KUKA KRL program: MyProgram_194().src

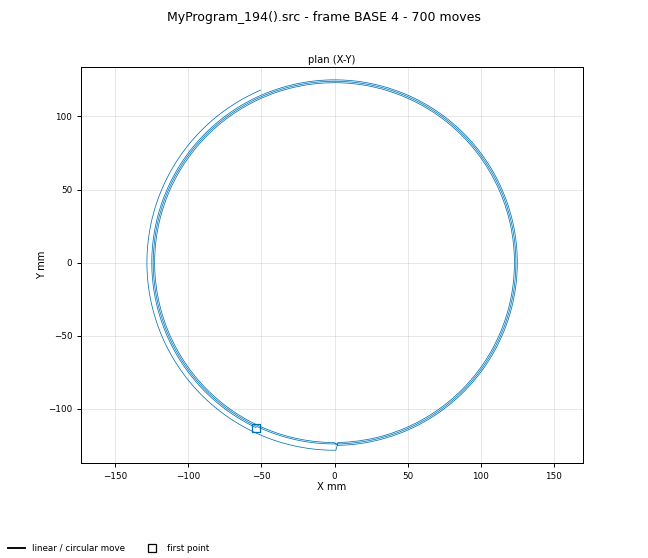
[picture p0: tool path of MyProgram_194().src in frame BASE 4, 700 of 700 moves have a stored position in this frame; points joined in program order, loops and branches not executed]
&ACCESS RVP
&REL 1
&PARAM TEMPLATE = C:\KRC\Roboter\Template\vorgabe
&PARAM EDITMASK = *
DEF MyProgram_194()
; ---- Setting reference (Base) ----
$BASE = BASE_DATA[4]

; --------------------------
; ---- Setting tool (TCP) ----
$TOOL = TOOL_DATA[3]
; --------------------------

$VEL.CP = VEL_APROX_PRINT
Startdeposition()
$VEL.CP = VEL_PRINT
LIN {X -53.6919,Y -112.9399,Z 140,A -118.7659,B 24.3079,C -1.2792,E1 24.2705,E2 205.3215} C_DIS
LIN {X -56.5912,Y -111.5152,Z 140,A -120.1079,B 24.3075,C -1.2873,E1 24.2671,E2 206.6473} C_DIS
LIN {X -59.8719,Y -109.7908,Z 140,A -122.1119,B 24.3081,C -1.2756,E1 24.2621,E2 208.6856} C_DIS
LIN {X -63.0275,Y -108.0107,Z 140,A -124.4326,B 24.3094,C -1.2483,E1 24.2563,E2 211.08} C_DIS
LIN {X -67.2513,Y -105.4322,Z 140,A -126.1298,B 24.308,C -1.2774,E1 24.2525,E2 212.7119} C_DIS
LIN {X -70.1428,Y -103.5309,Z 140,A -127.4855,B 24.3074,C -1.2903,E1 24.2494,E2 214.0408} C_DIS
LIN {X -72.9333,Y -101.5847,Z 140,A -129.2817,B 24.3078,C -1.2823,E1 24.2452,E2 215.8629} C_DIS
LIN {X -76.3639,Y -99.0319,Z 140,A -131.2624,B 24.3076,C -1.2848,E1 24.2408,E2 217.8448} C_DIS
LIN {X -79.5467,Y -96.4938,Z 140,A -133.1846,B 24.3076,C -1.2858,E1 24.2366,E2 219.7721} C_DIS
LIN {X -83.0381,Y -93.5062,Z 140,A -135.2359,B 24.3072,C -1.2924,E1 24.2323,E2 221.8156} C_DIS
LIN {X -86.157,Y -90.6407,Z 140,A -137.2143,B 24.3072,C -1.2947,E1 24.2283,E2 223.7967} C_DIS
LIN {X -89.322,Y -87.5228,Z 140,A -139.2228,B 24.3069,C -1.3003,E1 24.2243,E2 225.8004} C_DIS
LIN {X -91.6108,Y -85.1243,Z 140,A -140.6773,B 24.3065,C -1.3065,E1 24.2216,E2 227.2461} C_DIS
LIN {X -95.1006,Y -81.2071,Z 140,A -143.1881,B 24.3065,C -1.3073,E1 24.2169,E2 229.7666} C_DIS
LIN {X -97.6117,Y -78.1712,Z 140,A -145.009,B 24.3063,C -1.311,E1 24.2137,E2 231.5874} C_DIS
LIN {X -100.1442,Y -74.8991,Z 140,A -146.9149,B 24.3061,C -1.3152,E1 24.2105,E2 233.4924} C_DIS
LIN {X -102.2447,Y -72.0048,Z 140,A -148.8726,B 24.3066,C -1.3054,E1 24.2073,E2 235.4839} C_DIS
LIN {X -104.3595,Y -68.9041,Z 140,A -150.5706,B 24.3063,C -1.3108,E1 24.2047,E2 237.1775} C_DIS
LIN {X -106.3024,Y -65.8673,Z 140,A -151.9331,B 24.3055,C -1.3278,E1 24.2027,E2 238.5057} C_DIS
LIN {X -108.4877,Y -62.2025,Z 140,A -153.9183,B 24.3053,C -1.3317,E1 24.1999,E2 240.4918} C_DIS
LIN {X -110.5462,Y -58.4624,Z 140,A -155.833,B 24.3049,C -1.339,E1 24.1974,E2 242.3992} C_DIS
LIN {X -112.655,Y -54.2883,Z 140,A -158.0264,B 24.3047,C -1.3428,E1 24.1947,E2 244.5954} C_DIS
LIN {X -113.9621,Y -51.4883,Z 140,A -159.552,B 24.3047,C -1.3421,E1 24.1929,E2 246.1313} C_DIS
LIN {X -115.8635,Y -47.0528,Z 140,A -161.597,B 24.304,C -1.3558,E1 24.1907,E2 248.1546} C_DIS
LIN {X -117.0482,Y -44.0221,Z 140,A -163.0377,B 24.3037,C -1.3624,E1 24.1893,E2 249.5876} C_DIS
LIN {X -118.0271,Y -41.3277,Z 140,A -164.4301,B 24.3037,C -1.3629,E1 24.188,E2 250.9868} C_DIS
LIN {X -119.0708,Y -38.2151,Z 140,A -165.9048,B 24.3033,C -1.3688,E1 24.1867,E2 252.456} C_DIS
LIN {X -120.7278,Y -32.6066,Z 140,A -168.6751,B 24.3031,C -1.3731,E1 24.1845,E2 255.2322} C_DIS
LIN {X -121.683,Y -28.8394,Z 140,A -171.0654,B 24.3042,C -1.3525,E1 24.183,E2 257.6873} C_DIS
LIN {X -122.7191,Y -24.0546,Z 140,A -172.5557,B 24.3021,C -1.3918,E1 24.1822,E2 259.0906} C_DIS
LIN {X -123.7321,Y -18.1343,Z 140,A -175.4845,B 24.3021,C -1.3929,E1 24.1808,E2 262.0347} C_DIS
LIN {X -124.1912,Y -14.6583,Z 140,A -177.2858,B 24.3022,C -1.3897,E1 24.1802,E2 263.8548} C_DIS
LIN {X -124.6891,Y -9.5463,Z 140,A -179.4863,B 24.3014,C -1.4038,E1 24.1797,E2 266.0345} C_DIS
LIN {X -124.93,Y -5.5935,Z 140,A 178.647,B 24.3012,C -1.4075,E1 24.1794,E2 267.9039} C_DIS
LIN {X -125.0405,Y -1.8059,Z 140,A 177.1827,B 24.3003,C -1.4248,E1 24.1793,E2 269.3348} C_DIS
LIN {X -125.0536,Y 0.6006,Z 140,A 175.2536,B 24.302,C -1.3931,E1 24.1793,E2 271.3536} C_DIS
LIN {X -124.9418,Y 5.2951,Z 140,A 173.618,B 24.3004,C -1.4221,E1 24.1795,E2 272.9285} C_DIS
LIN {X -124.7099,Y 9.2612,Z 140,A 171.2259,B 24.3014,C -1.4037,E1 24.18,E2 275.3803} C_DIS
LIN {X -124.2464,Y 14.1956,Z 140,A 169.6952,B 24.2993,C -1.4426,E1 24.1804,E2 276.8253} C_DIS
LIN {X -123.3534,Y 20.5476,Z 140,A 166.6428,B 24.299,C -1.4473,E1 24.1817,E2 279.8851} C_DIS
LIN {X -122.8031,Y 23.6152,Z 140,A 165.0229,B 24.2992,C -1.4437,E1 24.1825,E2 281.5236} C_DIS
LIN {X -121.7214,Y 28.6802,Z 140,A 162.7251,B 24.2986,C -1.4545,E1 24.1839,E2 283.8089} C_DIS
LIN {X -120.7968,Y 32.3479,Z 140,A 161.1059,B 24.2981,C -1.465,E1 24.185,E2 285.4122} C_DIS
LIN {X -119.8901,Y 35.5638,Z 140,A 159.5609,B 24.2978,C -1.4692,E1 24.1862,E2 286.956} C_DIS
LIN {X -118.4982,Y 39.9577,Z 140,A 157.3573,B 24.2977,C -1.472,E1 24.1881,E2 289.166} C_DIS
LIN {X -117.1953,Y 43.6296,Z 140,A 155.618,B 24.2972,C -1.4795,E1 24.1897,E2 290.8969} C_DIS
LIN {X -115.9948,Y 46.7269,Z 140,A 153.9199,B 24.2974,C -1.4767,E1 24.1915,E2 292.6117} C_DIS
LIN {X -114.7571,Y 49.6891,Z 140,A 152.2718,B 24.2976,C -1.4736,E1 24.1934,E2 294.2767} C_DIS
LIN {X -113.4363,Y 52.6348,Z 140,A 150.9968,B 24.2968,C -1.4869,E1 24.1948,E2 295.5265} C_DIS
LIN {X -111.6462,Y 56.3339,Z 140,A 149.1355,B 24.2964,C -1.4934,E1 24.1971,E2 297.3821} C_DIS
LIN {X -110.3342,Y 58.8656,Z 140,A 147.8595,B 24.2961,C -1.4986,E1 24.1988,E2 298.6525} C_DIS
LIN {X -108.0224,Y 63.0061,Z 140,A 145.4957,B 24.2962,C -1.4968,E1 24.2021,E2 301.0336} C_DIS
LIN {X -105.5652,Y 67.043,Z 140,A 143.405,B 24.2957,C -1.5062,E1 24.2051,E2 303.1123} C_DIS
LIN {X -103.2652,Y 70.5339,Z 140,A 141.529,B 24.2953,C -1.5133,E1 24.208,E2 304.9806} C_DIS
LIN {X -101.1094,Y 73.5907,Z 140,A 139.7773,B 24.2951,C -1.5164,E1 24.2109,E2 306.7335} C_DIS
LIN {X -98.532,Y 77.0078,Z 140,A 137.7937,B 24.2948,C -1.5207,E1 24.2143,E2 308.7163} C_DIS
LIN {X -95.8068,Y 80.3723,Z 140,A 135.8162,B 24.2945,C -1.5262,E1 24.2178,E2 310.6897} C_DIS
LIN {X -92.9689,Y 83.6392,Z 140,A 133.8174,B 24.2942,C -1.5306,E1 24.2214,E2 312.6871} C_DIS
LIN {X -90.0744,Y 86.7489,Z 140,A 131.8247,B 24.2941,C -1.5334,E1 24.2253,E2 314.6818} C_DIS
LIN {X -86.8221,Y 90.0035,Z 140,A 129.7974,B 24.2936,C -1.5421,E1 24.2293,E2 316.6968} C_DIS
LIN {X -83.7569,Y 92.8632,Z 140,A 127.7843,B 24.2936,C -1.5425,E1 24.2334,E2 318.7171} C_DIS
LIN {X -80.5197,Y 95.6832,Z 140,A 125.8611,B 24.2932,C -1.5489,E1 24.2375,E2 320.6324} C_DIS
LIN {X -77.3248,Y 98.2829,Z 140,A 123.9446,B 24.293,C -1.5518,E1 24.2417,E2 322.5494} C_DIS
LIN {X -73.8783,Y 100.8994,Z 140,A 121.9198,B 24.2928,C -1.5541,E1 24.2462,E2 324.576} C_DIS
LIN {X -70.4181,Y 103.3445,Z 140,A 119.9558,B 24.2927,C -1.557,E1 24.2507,E2 326.5399} C_DIS
LIN {X -66.6736,Y 105.7984,Z 140,A 117.95,B 24.2923,C -1.5629,E1 24.2554,E2 328.5378} C_DIS
LIN {X -63.9124,Y 107.489,Z 140,A 116.1645,B 24.293,C -1.5524,E1 24.2598,E2 330.3547} C_DIS
LIN {X -60.9161,Y 109.2142,Z 140,A 114.5683,B 24.2928,C -1.5546,E1 24.2637,E2 331.9502} C_DIS
LIN {X -57.8736,Y 110.8554,Z 140,A 113.5124,B 24.2912,C -1.5807,E1 24.2661,E2 332.9456} C_DIS
LIN {X -54.8742,Y 112.3711,Z 140,A 111.3515,B 24.2928,C -1.5556,E1 24.2717,E2 335.1734} C_DIS
LIN {X -51.3522,Y 114.023,Z 140,A 109.9613,B 24.2915,C -1.5757,E1 24.2751,E2 336.5181} C_DIS
LIN {X -47.4788,Y 115.6917,Z 140,A 107.9839,B 24.2915,C -1.5764,E1 24.2802,E2 338.4984} C_DIS
LIN {X -44.6099,Y 116.8278,Z 140,A 106.6024,B 24.2913,C -1.5798,E1 24.2838,E2 339.8748} C_DIS
LIN {X -41.6192,Y 117.9259,Z 140,A 104.3148,B 24.2934,C -1.5449,E1 24.2901,E2 342.252} C_DIS
LIN {X -35.9049,Y 119.7898,Z 140,A 102.3187,B 24.2912,C -1.5817,E1 24.2952,E2 344.1621} C_DIS
LIN {X -32.8305,Y 120.6681,Z 140,A 100.5146,B 24.292,C -1.568,E1 24.3001,E2 346.0023} C_DIS
LIN {X -29.118,Y 121.6159,Z 140,A 98.6999,B 24.292,C -1.567,E1 24.3051,E2 347.822} C_DIS
LIN {X -25.0294,Y 122.5226,Z 140,A 97.2935,B 24.2906,C -1.5917,E1 24.3088,E2 349.1699} C_DIS
LIN {X -21.6294,Y 123.169,Z 140,A 95.5831,B 24.2908,C -1.5873,E1 24.3135,E2 350.893} C_DIS
LIN {X -17.7649,Y 123.7849,Z 140,A 93.8925,B 24.2905,C -1.5931,E1 24.3181,E2 352.5708} C_DIS
LIN {X -13.8843,Y 124.281,Z 140,A 92.0908,B 24.2905,C -1.5937,E1 24.3231,E2 354.3723} C_DIS
LIN {X -10.2183,Y 124.6354,Z 140,A 90.3228,B 24.2906,C -1.5909,E1 24.328,E2 356.1481} C_DIS
LIN {X -6.2274,Y 124.8981,Z 140,A 88.5896,B 24.2903,C -1.5961,E1 24.3328,E2 357.8691} C_DIS
LIN {X -2.719,Y 125.0254,Z 140,A 86.9015,B 24.2905,C -1.5929,E1 24.3376,E2 359.5653} C_DIS
LIN {X 1.0171,Y 125.0496,Z 140,A 85.1762,B 24.2905,C -1.5926,E1 24.3424,E2 361.2912} C_DIS
LIN {X 4.9283,Y 124.9561,Z 140,A 83.4543,B 24.2903,C -1.596,E1 24.3472,E2 363.0044} C_DIS
LIN {X 8.9204,Y 124.7348,Z 140,A 81.6298,B 24.2903,C -1.5964,E1 24.3523,E2 364.8273} C_DIS
LIN {X 12.4955,Y 124.4285,Z 140,A 79.8894,B 24.2906,C -1.5917,E1 24.3571,E2 366.5781} C_DIS
LIN {X 16.3314,Y 123.9821,Z 140,A 78.2129,B 24.2903,C -1.5956,E1 24.3617,E2 368.2436} C_DIS
LIN {X 20.3658,Y 123.3838,Z 140,A 76.3517,B 24.2903,C -1.5954,E1 24.3669,E2 370.1036} C_DIS
LIN {X 24.186,Y 122.694,Z 140,A 74.372,B 24.291,C -1.5853,E1 24.3724,E2 372.1055} C_DIS
LIN {X 29.3374,Y 121.563,Z 140,A 72.182,B 24.2904,C -1.5946,E1 24.3783,E2 374.2698} C_DIS
LIN {X 32.964,Y 120.6323,Z 140,A 70.3195,B 24.2909,C -1.5865,E1 24.3833,E2 376.1488} C_DIS
LIN {X 36.874,Y 119.4932,Z 140,A 68.5454,B 24.2907,C -1.5894,E1 24.388,E2 377.9126} C_DIS
LIN {X 40.4587,Y 118.3283,Z 140,A 66.9207,B 24.2905,C -1.5928,E1 24.3923,E2 379.526} C_DIS
LIN {X 43.1079,Y 117.3901,Z 140,A 65.0136,B 24.2923,C -1.5624,E1 24.3975,E2 381.5026} C_DIS
LIN {X 47.2438,Y 115.7865,Z 140,A 63.4562,B 24.2911,C -1.5827,E1 24.4014,E2 383.0074} C_DIS
LIN {X 50.698,Y 114.3156,Z 140,A 61.8125,B 24.2911,C -1.5844,E1 24.4056,E2 384.6428} C_DIS
LIN {X 54.3579,Y 112.6217,Z 140,A 59.6104,B 24.2922,C -1.5653,E1 24.4112,E2 386.8852} C_DIS
LIN {X 57.603,Y 110.9975,Z 140,A 58.2793,B 24.2913,C -1.5788,E1 24.4145,E2 388.1797} C_DIS
LIN {X 63.6338,Y 107.6546,Z 140,A 55.1206,B 24.2916,C -1.5743,E1 24.4222,E2 391.3398} C_DIS
LIN {X 67.1422,Y 105.5021,Z 140,A 53.3746,B 24.2914,C -1.578,E1 24.4262,E2 393.0709} C_DIS
LIN {X 70.2121,Y 103.484,Z 140,A 51.6783,B 24.2916,C -1.5746,E1 24.4302,E2 394.7697} C_DIS
LIN {X 73.1481,Y 101.4302,Z 140,A 50.0018,B 24.2919,C -1.5701,E1 24.434,E2 396.4511} C_DIS
LIN {X 76.1718,Y 99.1795,Z 140,A 48.3051,B 24.2919,C -1.5685,E1 24.4378,E2 398.1456} C_DIS
LIN {X 80.5194,Y 95.6834,Z 140,A 45.661,B 24.2925,C -1.5593,E1 24.4436,E2 400.8015} C_DIS
LIN {X 83.7682,Y 92.8529,Z 140,A 43.6395,B 24.2929,C -1.553,E1 24.4478,E2 402.8298} C_DIS
LIN {X 87.085,Y 89.7489,Z 140,A 41.6152,B 24.293,C -1.5514,E1 24.4519,E2 404.8495} C_DIS
LIN {X 90.0335,Y 86.7911,Z 140,A 39.6982,B 24.2933,C -1.547,E1 24.4556,E2 406.7686} C_DIS
LIN {X 92.8649,Y 83.755,Z 140,A 37.7842,B 24.2936,C -1.5421,E1 24.4592,E2 408.6858} C_DIS
LIN {X 95.6504,Y 80.5588,Z 140,A 35.8982,B 24.2936,C -1.5403,E1 24.4627,E2 410.5672} C_DIS
LIN {X 98.1158,Y 77.5376,Z 140,A 34.0944,B 24.294,C -1.5352,E1 24.4658,E2 412.3749} C_DIS
LIN {X 100.6643,Y 74.1983,Z 140,A 32.3122,B 24.2938,C -1.5374,E1 24.4688,E2 414.1431} C_DIS
LIN {X 103.2862,Y 70.5033,Z 140,A 30.1538,B 24.2944,C -1.528,E1 24.4723,E2 416.3133} C_DIS
LIN {X 105.5787,Y 67.0216,Z 140,A 28.1882,B 24.2949,C -1.5202,E1 24.4753,E2 418.2874} C_DIS
LIN {X 107.2835,Y 64.2572,Z 140,A 26.4298,B 24.2959,C -1.5029,E1 24.4778,E2 420.0784} C_DIS
LIN {X 109.1198,Y 61.0865,Z 140,A 25.055,B 24.2953,C -1.5132,E1 24.4797,E2 421.4208} C_DIS
LIN {X 110.6437,Y 58.2767,Z 140,A 23.1393,B 24.2968,C -1.487,E1 24.4822,E2 423.3896} C_DIS
LIN {X 112.6736,Y 54.2493,Z 140,A 21.7292,B 24.2953,C -1.5134,E1 24.4839,E2 424.728} C_DIS
LIN {X 114.1511,Y 51.0659,Z 140,A 20.0748,B 24.2957,C -1.5065,E1 24.4858,E2 426.3899} C_DIS
LIN {X 115.3595,Y 48.2741,Z 140,A 18.7408,B 24.2957,C -1.5054,E1 24.4873,E2 427.7191} C_DIS
LIN {X 116.3256,Y 45.9017,Z 140,A 17.4038,B 24.2964,C -1.4938,E1 24.4887,E2 429.0764} C_DIS
LIN {X 117.9032,Y 41.6849,Z 140,A 14.9511,B 24.2979,C -1.4683,E1 24.491,E2 431.5767} C_DIS
LIN {X 119.1859,Y 37.8547,Z 140,A 13.4947,B 24.2971,C -1.4822,E1 24.4922,E2 432.991} C_DIS
LIN {X 120.8839,Y 32.0214,Z 140,A 10.8374,B 24.2972,C -1.4799,E1 24.4943,E2 435.6381} C_DIS
LIN {X 121.8046,Y 28.3208,Z 140,A 9.1135,B 24.2974,C -1.4756,E1 24.4954,E2 437.3621} C_DIS
LIN {X 122.5443,Y 24.923,Z 140,A 7.5415,B 24.2977,C -1.4716,E1 24.4963,E2 438.9342} C_DIS
LIN {X 123.2508,Y 21.1628,Z 140,A 5.724,B 24.2982,C -1.4628,E1 24.4972,E2 440.7621} C_DIS
LIN {X 123.8051,Y 17.6236,Z 140,A 4.1393,B 24.2983,C -1.4604,E1 24.4978,E2 442.343} C_DIS
LIN {X 124.3134,Y 13.5837,Z 140,A 2.3029,B 24.2986,C -1.4558,E1 24.4985,E2 444.1792} C_DIS
LIN {X 124.6751,Y 9.7384,Z 140,A 0.4725,B 24.2991,C -1.447,E1 24.4989,E2 446.0197} C_DIS
LIN {X 124.9132,Y 5.9267,Z 140,A -1.2863,B 24.2994,C -1.4409,E1 24.4992,E2 447.7825} C_DIS
LIN {X 125.0374,Y 1.9942,Z 140,A -2.9417,B 24.2994,C -1.4424,E1 24.4992,E2 449.4241} C_DIS
LIN {X 125.0322,Y -2.3088,Z 140,A -5.0331,B 24.3,C -1.43,E1 24.4992,E2 451.5328} C_DIS
LIN {X 124.8915,Y -6.358,Z 140,A -6.7859,B 24.3,C -1.4291,E1 24.499,E2 453.2769} C_DIS
LIN {X 124.6624,Y -9.8989,Z 140,A -8.4794,B 24.3005,C -1.4203,E1 24.4987,E2 454.9812} C_DIS
LIN {X 124.3069,Y -13.644,Z 140,A -10.2178,B 24.3009,C -1.414,E1 24.4982,E2 456.7244} C_DIS
LIN {X 123.7958,Y -17.688,Z 140,A -11.9726,B 24.3009,C -1.4135,E1 24.4975,E2 458.4695} C_DIS
LIN {X 123.1515,Y -21.7273,Z 140,A -13.8398,B 24.3012,C -1.4078,E1 24.4967,E2 460.3394} C_DIS
LIN {X 121.8901,Y -27.9473,Z 140,A -17.1147,B 24.3027,C -1.38,E1 24.4947,E2 463.6617} C_DIS
LIN {X 120.9852,Y -31.6414,Z 140,A -18.357,B 24.3017,C -1.3994,E1 24.4939,E2 464.8498} C_DIS
LIN {X 120.1853,Y -34.5514,Z 140,A -20.0597,B 24.3028,C -1.379,E1 24.4926,E2 466.5918} C_DIS
LIN {X 118.7173,Y -39.2996,Z 140,A -22.4113,B 24.3034,C -1.368,E1 24.4906,E2 468.9561} C_DIS
LIN {X 117.6172,Y -42.4784,Z 140,A -23.603,B 24.3027,C -1.3806,E1 24.4895,E2 470.1105} C_DIS
LIN {X 116.369,Y -45.79,Z 140,A -25.192,B 24.3029,C -1.3772,E1 24.4879,E2 471.6988} C_DIS
LIN {X 115.0127,Y -49.098,Z 140,A -26.9146,B 24.3034,C -1.3678,E1 24.486,E2 473.4341} C_DIS
LIN {X 112.0407,Y -55.544,Z 140,A -30.0975,B 24.3037,C -1.3614,E1 24.4822,E2 476.6149} C_DIS
LIN {X 109.9969,Y -59.4933,Z 140,A -32.1786,B 24.3041,C -1.3531,E1 24.4795,E2 478.7047} C_DIS
LIN {X 108.034,Y -62.9877,Z 140,A -34.0489,B 24.3045,C -1.346,E1 24.4769,E2 480.5823} C_DIS
LIN {X 105.6721,Y -66.8737,Z 140,A -36.0672,B 24.3047,C -1.3432,E1 24.4739,E2 482.5967} C_DIS
LIN {X 102.7414,Y -71.2944,Z 140,A -38.3754,B 24.3047,C -1.3424,E1 24.4704,E2 484.8951} C_DIS
LIN {X 100.5448,Y -74.361,Z 140,A -40.2595,B 24.3054,C -1.3298,E1 24.4672,E2 486.8001} C_DIS
LIN {X 97.8823,Y -77.8313,Z 140,A -42.2174,B 24.3055,C -1.3267,E1 24.4639,E2 488.7562} C_DIS
LIN {X 94.2467,Y -82.1962,Z 140,A -44.7886,B 24.3058,C -1.3214,E1 24.4592,E2 491.328} C_DIS
LIN {X 89.1498,Y -87.6983,Z 140,A -48.0245,B 24.3058,C -1.3226,E1 24.4531,E2 494.5465} C_DIS
LIN {X 85.4413,Y -91.3155,Z 140,A -50.5983,B 24.3065,C -1.3069,E1 24.4478,E2 497.1472} C_DIS
LIN {X 80.2995,Y -95.8679,Z 140,A -53.7377,B 24.3069,C -1.3,E1 24.4412,E2 500.2906} C_DIS
LIN {X 76.9147,Y -98.6049,Z 140,A -55.7259,B 24.3071,C -1.2959,E1 24.4369,E2 502.2812} C_DIS
LIN {X 73.3148,Y -101.3095,Z 140,A -57.4223,B 24.3064,C -1.3095,E1 24.4332,E2 503.9382} C_DIS
LIN {X 68.4944,Y -104.6293,Z 140,A -60.4164,B 24.3074,C -1.2887,E1 24.4262,E2 506.9722} C_DIS
LIN {X 64.8243,Y -106.9415,Z 140,A -62.3627,B 24.3075,C -1.2869,E1 24.4215,E2 508.9166} C_DIS
LIN {X 61.0777,Y -109.1248,Z 140,A -64.375,B 24.3078,C -1.2821,E1 24.4166,E2 510.9344} C_DIS
LIN {X 57.1048,Y -111.2538,Z 140,A -66.3773,B 24.3078,C -1.2816,E1 24.4117,E2 512.9321} C_DIS
LIN {X 54.2085,Y -112.6931,Z 140,A -67.7822,B 24.3078,C -1.2829,E1 24.4082,E2 514.3299} C_DIS
LIN {X 51.3542,Y -114.0221,Z 140,A -69.338,B 24.3081,C -1.2752,E1 24.4042,E2 515.9004} C_DIS
LIN {X 47.6413,Y -115.6238,Z 140,A -71.2144,B 24.3083,C -1.2713,E1 24.3994,E2 517.7817} C_DIS
LIN {X 44.1737,Y -116.9914,Z 140,A -73.5929,B 24.31,C -1.2368,E1 24.393,E2 520.2386} C_DIS
LIN {X 38.856,Y -118.865,Z 140,A -75.3361,B 24.3082,C -1.2737,E1 24.3886,E2 521.8887} C_DIS
LIN {X 32.1785,Y -120.842,Z 140,A -78.5471,B 24.3084,C -1.2691,E1 24.38,E2 525.1052} C_DIS
LIN {X 28.7784,Y -121.6977,Z 140,A -80.1455,B 24.3084,C -1.2679,E1 24.3756,E2 526.7042} C_DIS
LIN {X 24.9652,Y -122.5357,Z 140,A -81.941,B 24.3086,C -1.266,E1 24.3707,E2 528.502} C_DIS
LIN {X 21.4154,Y -123.2073,Z 140,A -83.6474,B 24.3087,C -1.2622,E1 24.366,E2 530.2157} C_DIS
LIN {X 17.7573,Y -123.7859,Z 140,A -85.2968,B 24.3087,C -1.2633,E1 24.3615,E2 531.8608} C_DIS
LIN {X 14.0315,Y -124.2652,Z 140,A -87.0869,B 24.3089,C -1.2589,E1 24.3565,E2 533.6602} C_DIS
LIN {X 10.4122,Y -124.619,Z 140,A -88.6895,B 24.3088,C -1.2611,E1 24.352,E2 535.2565} C_DIS
LIN {X 6.4833,Y -124.8852,Z 140,A -90.5192,B 24.3088,C -1.2591,E1 24.3469,E2 537.0903} C_DIS
LIN {X 2.4731,Y -125.0294,Z 140,A -92.3766,B 24.309,C -1.2576,E1 24.3417,E2 538.9509} C_DIS
LIN {X 2.4731,Y -125.0294,Z 140,A -92.3766,B 24.309,C -1.2576,E1 24.3417,E2 538.9509} C_DIS
Enddeposition()
LIN {X 0.8758,Y -124.0739,Z 140,A -92.8769,B 23.7005,C -1.164,E1 23.7279,E2 539.5997} C_DIS
Startdeposition()
$VEL.CP = VEL_PRINT
LIN {X 5.1874,Y -123.9703,Z 140,A -90.2212,B 23.6991,C -1.195,E1 23.7355,E2 536.8673} C_DIS
LIN {X 8.9976,Y -123.7516,Z 140,A -88.3652,B 23.6989,C -1.2001,E1 23.7407,E2 534.9995} C_DIS
LIN {X 13.0801,Y -123.387,Z 140,A -86.5046,B 23.6989,C -1.1996,E1 23.7459,E2 533.1412} C_DIS
LIN {X 16.4159,Y -122.9878,Z 140,A -84.9017,B 23.6987,C -1.203,E1 23.7503,E2 531.5313} C_DIS
LIN {X 20.3643,Y -122.3956,Z 140,A -83.1274,B 23.6988,C -1.2011,E1 23.7552,E2 529.7636} C_DIS
LIN {X 23.38,Y -121.8554,Z 140,A -81.6488,B 23.6986,C -1.2053,E1 23.7593,E2 528.2764} C_DIS
LIN {X 27.1976,Y -121.0613,Z 140,A -79.4825,B 23.6977,C -1.2241,E1 23.7653,E2 526.0664} C_DIS
LIN {X 30.9893,Y -120.1468,Z 140,A -78.0716,B 23.6985,C -1.2075,E1 23.769,E2 524.699} C_DIS
LIN {X 38.5918,Y -117.9254,Z 140,A -74.5759,B 23.6987,C -1.204,E1 23.7783,E2 521.2185} C_DIS
LIN {X 43.8221,Y -116.0821,Z 140,A -71.9287,B 23.6983,C -1.2115,E1 23.7853,E2 518.5586} C_DIS
LIN {X 46.5763,Y -115.0043,Z 140,A -70.4957,B 23.6981,C -1.2166,E1 23.789,E2 517.1163} C_DIS
LIN {X 49.8037,Y -113.6454,Z 140,A -69.0055,B 23.6982,C -1.2129,E1 23.7928,E2 515.639} C_DIS
LIN {X 52.648,Y -112.356,Z 140,A -67.5899,B 23.6982,C -1.2139,E1 23.7964,E2 514.2247} C_DIS
LIN {X 55.0194,Y -111.2123,Z 140,A -66.3236,B 23.698,C -1.2183,E1 23.7996,E2 512.951} C_DIS
LIN {X 58.3255,Y -109.5169,Z 140,A -64.508,B 23.6976,C -1.226,E1 23.8041,E2 511.1218} C_DIS
LIN {X 61.5286,Y -107.7497,Z 140,A -62.8692,B 23.6976,C -1.2266,E1 23.8081,E2 509.4866} C_DIS
LIN {X 64.6525,Y -105.9051,Z 140,A -61.2958,B 23.6976,C -1.2248,E1 23.8119,E2 507.9229} C_DIS
LIN {X 67.6259,Y -104.0312,Z 140,A -59.657,B 23.6975,C -1.2287,E1 23.8157,E2 506.2801} C_DIS
LIN {X 71.3355,Y -101.5236,Z 140,A -57.7263,B 23.6975,C -1.2263,E1 23.8202,E2 504.3623} C_DIS
LIN {X 73.7735,Y -99.7666,Z 140,A -56.07,B 23.6968,C -1.2421,E1 23.824,E2 502.673} C_DIS
LIN {X 77.3218,Y -97.0418,Z 140,A -54.0651,B 23.6968,C -1.2437,E1 23.8284,E2 500.6721} C_DIS
LIN {X 80.6334,Y -94.3082,Z 140,A -52.0635,B 23.6965,C -1.2491,E1 23.8326,E2 498.6653} C_DIS
LIN {X 82.9928,Y -92.239,Z 140,A -50.6939,B 23.6965,C -1.2486,E1 23.8355,E2 497.3027} C_DIS
LIN {X 86.0033,Y -89.4389,Z 140,A -48.7547,B 23.6962,C -1.2551,E1 23.8394,E2 495.356} C_DIS
LIN {X 89.6603,Y -85.7716,Z 140,A -46.2997,B 23.6957,C -1.2641,E1 23.8442,E2 492.8898} C_DIS
LIN {X 91.9569,Y -83.3048,Z 140,A -44.8695,B 23.6958,C -1.2619,E1 23.8469,E2 491.4717} C_DIS
LIN {X 94.4731,Y -80.44,Z 140,A -43.0875,B 23.6955,C -1.2675,E1 23.8502,E2 489.6843} C_DIS
LIN {X 97.9235,Y -76.2024,Z 140,A -40.7829,B 23.6957,C -1.2636,E1 23.8542,E2 487.4009} C_DIS
LIN {X 99.712,Y -73.847,Z 140,A -39.363,B 23.6954,C -1.2699,E1 23.8566,E2 485.9725} C_DIS
LIN {X 101.7025,Y -71.0805,Z 140,A -37.6313,B 23.6948,C -1.282,E1 23.8594,E2 484.2198} C_DIS
LIN {X 103.8864,Y -67.849,Z 140,A -35.8252,B 23.6945,C -1.2873,E1 23.8622,E2 482.4101} C_DIS
LIN {X 106.1614,Y -64.2301,Z 140,A -33.964,B 23.6945,C -1.2875,E1 23.8649,E2 480.5584} C_DIS
LIN {X 108.1442,Y -60.8325,Z 140,A -32.0915,B 23.6941,C -1.2956,E1 23.8675,E2 478.6763} C_DIS
LIN {X 110.0019,Y -57.4018,Z 140,A -30.3709,B 23.6941,C -1.297,E1 23.8698,E2 476.9618} C_DIS
LIN {X 112.2352,Y -52.9053,Z 140,A -28.1101,B 23.6938,C -1.3011,E1 23.8725,E2 474.7037} C_DIS
LIN {X 113.4448,Y -50.2572,Z 140,A -26.8255,B 23.6938,C -1.3023,E1 23.874,E2 473.4236} C_DIS
LIN {X 114.84,Y -46.9841,Z 140,A -25.2021,B 23.6936,C -1.3064,E1 23.8757,E2 471.7995} C_DIS
LIN {X 115.7727,Y -44.633,Z 140,A -23.8604,B 23.6929,C -1.3185,E1 23.8771,E2 470.4356} C_DIS
LIN {X 117.0146,Y -41.2717,Z 140,A -22.2604,B 23.6928,C -1.321,E1 23.8786,E2 468.839} C_DIS
LIN {X 118.1823,Y -37.7925,Z 140,A -20.5905,B 23.6926,C -1.3251,E1 23.8801,E2 467.1689} C_DIS
LIN {X 119.6482,Y -32.863,Z 140,A -18.3162,B 23.6924,C -1.3277,E1 23.8818,E2 464.902} C_DIS
LIN {X 120.5452,Y -29.3992,Z 140,A -15.7166,B 23.6896,C -1.3799,E1 23.8836,E2 462.1891} C_DIS
LIN {X 121.8513,Y -23.4014,Z 140,A -14.1238,B 23.6924,C -1.3276,E1 23.8845,E2 460.7356} C_DIS
LIN {X 122.5522,Y -19.4042,Z 140,A -11.9092,B 23.6912,C -1.3504,E1 23.8855,E2 458.4786} C_DIS
LIN {X 123.0592,Y -15.871,Z 140,A -10.2349,B 23.6909,C -1.357,E1 23.8861,E2 456.7983} C_DIS
LIN {X 123.5013,Y -11.9511,Z 140,A -8.4609,B 23.6907,C -1.3606,E1 23.8866,E2 455.0266} C_DIS
LIN {X 123.7892,Y -8.4824,Z 140,A -6.8112,B 23.6903,C -1.3679,E1 23.887,E2 453.3692} C_DIS
LIN {X 123.9916,Y -4.6424,Z 140,A -5.0884,B 23.6901,C -1.3711,E1 23.8872,E2 451.6493} C_DIS
LIN {X 124.0798,Y -0.4469,Z 140,A -3.1978,B 23.6899,C -1.375,E1 23.8872,E2 449.761} C_DIS
LIN {X 124.0336,Y 3.3336,Z 140,A -1.5052,B 23.6897,C -1.3781,E1 23.8872,E2 448.0714} C_DIS
LIN {X 123.8785,Y 7.06,Z 140,A 0.3015,B 23.6892,C -1.3878,E1 23.8869,E2 446.2521} C_DIS
LIN {X 123.596,Y 10.9398,Z 140,A 1.9347,B 23.6893,C -1.3856,E1 23.8865,E2 444.6346} C_DIS
LIN {X 123.3449,Y 13.4712,Z 140,A 3.2481,B 23.6887,C -1.3962,E1 23.8862,E2 443.3034} C_DIS
LIN {X 122.8463,Y 17.4409,Z 140,A 4.9879,B 23.6887,C -1.3968,E1 23.8855,E2 441.5729} C_DIS
LIN {X 122.3231,Y 20.7985,Z 140,A 6.6929,B 23.688,C -1.4084,E1 23.8847,E2 439.8498} C_DIS
LIN {X 121.5587,Y 24.8771,Z 140,A 8.4818,B 23.688,C -1.4082,E1 23.8838,E2 438.0724} C_DIS
LIN {X 120.0892,Y 31.2161,Z 140,A 12.7615,B 23.6839,C -1.4805,E1 23.8807,E2 433.64} C_DIS
LIN {X 117.8106,Y 38.9367,Z 140,A 15.2091,B 23.6869,C -1.429,E1 23.8788,E2 431.3345} C_DIS
LIN {X 116.7162,Y 42.1028,Z 140,A 16.7086,B 23.6867,C -1.4313,E1 23.8774,E2 429.8383} C_DIS
LIN {X 115.5615,Y 45.1763,Z 140,A 18.1595,B 23.6867,C -1.4327,E1 23.8759,E2 428.3926} C_DIS
LIN {X 114.4202,Y 47.9934,Z 140,A 19.5546,B 23.6865,C -1.4363,E1 23.8745,E2 426.9965} C_DIS
LIN {X 112.9128,Y 51.4439,Z 140,A 21.239,B 23.6863,C -1.4387,E1 23.8725,E2 425.3161} C_DIS
LIN {X 111.7219,Y 53.9798,Z 140,A 22.7655,B 23.6855,C -1.4537,E1 23.8707,E2 423.7611} C_DIS
LIN {X 110.2585,Y 56.9108,Z 140,A 24.1739,B 23.6855,C -1.4528,E1 23.8689,E2 422.3628} C_DIS
LIN {X 108.3276,Y 60.506,Z 140,A 25.993,B 23.6854,C -1.4548,E1 23.8665,E2 420.5489} C_DIS
LIN {X 106.3833,Y 63.8631,Z 140,A 27.5655,B 23.6857,C -1.4491,E1 23.8643,E2 418.9991} C_DIS
LIN {X 104.7689,Y 66.478,Z 140,A 29.2675,B 23.6847,C -1.4665,E1 23.8617,E2 417.2632} C_DIS
LIN {X 102.6594,Y 69.6909,Z 140,A 31.0162,B 23.6845,C -1.4698,E1 23.859,E2 415.5154} C_DIS
LIN {X 100.4653,Y 72.8181,Z 140,A 32.4906,B 23.6851,C -1.4604,E1 23.8566,E2 414.0721} C_DIS
LIN {X 98.8026,Y 75.0597,Z 140,A 34.0819,B 23.684,C -1.4781,E1 23.8539,E2 412.445} C_DIS
LIN {X 96.2657,Y 78.2864,Z 140,A 35.961,B 23.6838,C -1.4819,E1 23.8506,E2 410.5657} C_DIS
LIN {X 93.3484,Y 81.7427,Z 140,A 38.004,B 23.6837,C -1.4846,E1 23.8469,E2 408.5259} C_DIS
LIN {X 90.4707,Y 84.9171,Z 140,A 40.0094,B 23.6833,C -1.4903,E1 23.8431,E2 406.5156} C_DIS
LIN {X 87.5872,Y 87.8878,Z 140,A 41.8921,B 23.6832,C -1.4931,E1 23.8394,E2 404.6346} C_DIS
LIN {X 84.5624,Y 90.8017,Z 140,A 43.7994,B 23.683,C -1.4956,E1 23.8355,E2 402.7293} C_DIS
LIN {X 81.283,Y 93.7496,Z 140,A 45.8407,B 23.6827,C -1.4999,E1 23.8313,E2 400.686} C_DIS
LIN {X 77.5469,Y 96.8626,Z 140,A 48.1108,B 23.6824,C -1.5054,E1 23.8264,E2 398.4116} C_DIS
LIN {X 73.9177,Y 99.6594,Z 140,A 49.9855,B 23.6829,C -1.4978,E1 23.8222,E2 396.5628} C_DIS
LIN {X 71.204,Y 101.6164,Z 140,A 51.5508,B 23.6827,C -1.5014,E1 23.8187,E2 394.9943} C_DIS
LIN {X 68.6778,Y 103.3401,Z 140,A 53.1628,B 23.682,C -1.5132,E1 23.8149,E2 393.3589} C_DIS
LIN {X 66.0693,Y 105.0269,Z 140,A 54.5611,B 23.682,C -1.5137,E1 23.8116,E2 391.964} C_DIS
LIN {X 62.3969,Y 107.2495,Z 140,A 56.6502,B 23.6814,C -1.5217,E1 23.8065,E2 389.8619} C_DIS
LIN {X 58.4964,Y 109.4258,Z 140,A 58.6106,B 23.6816,C -1.5198,E1 23.8018,E2 387.9123} C_DIS
LIN {X 55.0433,Y 111.2005,Z 140,A 60.4056,B 23.6814,C -1.5222,E1 23.7973,E2 386.1164} C_DIS
LIN {X 50.6416,Y 113.2728,Z 140,A 62.4881,B 23.6817,C -1.5172,E1 23.792,E2 384.0519} C_DIS
LIN {X 47.1145,Y 114.7872,Z 140,A 64.2588,B 23.6817,C -1.519,E1 23.7875,E2 382.2811} C_DIS
LIN {X 43.2803,Y 116.285,Z 140,A 66.1666,B 23.6815,C -1.5213,E1 23.7825,E2 380.3722} C_DIS
LIN {X 40.5442,Y 117.2668,Z 140,A 67.5703,B 23.6812,C -1.5253,E1 23.7788,E2 378.9614} C_DIS
LIN {X 37.325,Y 118.3317,Z 140,A 69.0093,B 23.6815,C -1.5207,E1 23.775,E2 377.5367} C_DIS
LIN {X 34.2114,Y 119.2702,Z 140,A 70.5811,B 23.6812,C -1.525,E1 23.7708,E2 375.957} C_DIS
LIN {X 29.7652,Y 120.457,Z 140,A 73.4821,B 23.679,C -1.5622,E1 23.7627,E2 372.9683} C_DIS
LIN {X 24.5814,Y 121.6188,Z 140,A 74.8458,B 23.6819,C -1.5133,E1 23.7593,E2 371.7279} C_DIS
LIN {X 21.6856,Y 122.1685,Z 140,A 76.592,B 23.6808,C -1.5314,E1 23.7544,E2 369.9388} C_DIS
LIN {X 17.6497,Y 122.8165,Z 140,A 78.4103,B 23.681,C -1.5288,E1 23.7494,E2 368.1287} C_DIS
LIN {X 13.9338,Y 123.2951,Z 140,A 80.171,B 23.681,C -1.5306,E1 23.7445,E2 366.3651} C_DIS
LIN {X 10.2714,Y 123.6525,Z 140,A 81.8676,B 23.6809,C -1.5306,E1 23.7398,E2 364.6694} C_DIS
LIN {X 6.33,Y 123.9167,Z 140,A 83.6758,B 23.6809,C -1.53,E1 23.7347,E2 362.8637} C_DIS
LIN {X 2.4536,Y 124.0547,Z 140,A 85.5233,B 23.6808,C -1.5323,E1 23.7296,E2 361.0107} C_DIS
LIN {X -0.913,Y 124.0752,Z 140,A 86.9789,B 23.6811,C -1.5276,E1 23.7255,E2 359.5669} C_DIS
LIN {X -4.9295,Y 123.9804,Z 140,A 88.8773,B 23.681,C -1.529,E1 23.7202,E2 357.6647} C_DIS
LIN {X -8.9572,Y 123.7545,Z 140,A 90.7539,B 23.681,C -1.5289,E1 23.715,E2 355.7877} C_DIS
LIN {X -12.9891,Y 123.3968,Z 140,A 92.643,B 23.681,C -1.5289,E1 23.7097,E2 353.8976} C_DIS
LIN {X -17.0013,Y 122.9091,Z 140,A 94.431,B 23.6813,C -1.5242,E1 23.7048,E2 352.1198} C_DIS
LIN {X -20.3117,Y 122.4043,Z 140,A 96.017,B 23.6813,C -1.5249,E1 23.7004,E2 350.5305} C_DIS
LIN {X -23.8703,Y 121.7617,Z 140,A 97.6398,B 23.6814,C -1.5215,E1 23.696,E2 348.9144} C_DIS
LIN {X -27.3321,Y 121.0306,Z 140,A 99.4124,B 23.6812,C -1.5263,E1 23.6911,E2 347.1276} C_DIS
LIN {X -30.0273,Y 120.3909,Z 140,A 100.692,B 23.6812,C -1.5251,E1 23.6877,E2 345.8491} C_DIS
LIN {X -33.526,Y 119.4628,Z 140,A 102.2791,B 23.6816,C -1.5196,E1 23.6834,E2 344.273} C_DIS
LIN {X -36.8717,Y 118.4743,Z 140,A 103.8726,B 23.6817,C -1.5171,E1 23.6792,E2 342.6831} C_DIS
LIN {X -41.6439,Y 116.8817,Z 140,A 106.3119,B 23.6816,C -1.5193,E1 23.6727,E2 340.2332} C_DIS
LIN {X -45.2276,Y 115.5416,Z 140,A 107.9992,B 23.6819,C -1.5135,E1 23.6683,E2 338.5566} C_DIS
LIN {X -48.0112,Y 114.4127,Z 140,A 109.4262,B 23.6819,C -1.5133,E1 23.6646,E2 337.1267} C_DIS
LIN {X -51.9865,Y 112.6619,Z 140,A 111.893,B 23.6809,C -1.5304,E1 23.6582,E2 334.6108} C_DIS
LIN {X -55.7011,Y 110.8743,Z 140,A 113.2421,B 23.6826,C -1.5031,E1 23.655,E2 333.326} C_DIS
LIN {X -58.4183,Y 109.4677,Z 140,A 114.838,B 23.6822,C -1.5087,E1 23.651,E2 331.7115} C_DIS
LIN {X -62.2414,Y 107.3395,Z 140,A 117.1718,B 23.6816,C -1.5188,E1 23.6453,E2 329.3453} C_DIS
LIN {X -65.3722,Y 105.4622,Z 140,A 118.193,B 23.6835,C -1.4869,E1 23.6431,E2 328.4003} C_DIS
LIN {X -69.2537,Y 102.9554,Z 140,A 120.7332,B 23.6827,C -1.5003,E1 23.637,E2 325.8179} C_DIS
LIN {X -72.9133,Y 100.3963,Z 140,A 122.7752,B 23.683,C -1.4952,E1 23.6324,E2 323.781} C_DIS
LIN {X -76.3734,Y 97.7905,Z 140,A 124.7787,B 23.6833,C -1.4911,E1 23.628,E2 321.7801} C_DIS
LIN {X -79.6044,Y 95.1784,Z 140,A 126.6487,B 23.6836,C -1.4848,E1 23.6239,E2 319.9182} C_DIS
LIN {X -82.6141,Y 92.5781,Z 140,A 128.566,B 23.6836,C -1.4841,E1 23.6199,E2 317.9947} C_DIS
LIN {X -85.63,Y 89.7958,Z 140,A 130.4232,B 23.684,C -1.478,E1 23.6161,E2 316.1446} C_DIS
LIN {X -88.5419,Y 86.9258,Z 140,A 132.3506,B 23.6842,C -1.4751,E1 23.6123,E2 314.2158} C_DIS
LIN {X -91.615,Y 83.6816,Z 140,A 134.4524,B 23.6844,C -1.4716,E1 23.6083,E2 312.1131} C_DIS
LIN {X -94.3996,Y 80.5265,Z 140,A 136.3995,B 23.6847,C -1.4668,E1 23.6048,E2 310.1686} C_DIS
LIN {X -97.1698,Y 77.161,Z 140,A 138.3843,B 23.6851,C -1.4603,E1 23.6013,E2 308.1902} C_DIS
LIN {X -99.8003,Y 73.7277,Z 140,A 140.4504,B 23.6852,C -1.4578,E1 23.5978,E2 306.1199} C_DIS
LIN {X -102.3981,Y 70.0744,Z 140,A 142.5215,B 23.6856,C -1.4521,E1 23.5945,E2 304.0521} C_DIS
LIN {X -104.5764,Y 66.7799,Z 140,A 144.3147,B 23.6859,C -1.4457,E1 23.5918,E2 302.2655} C_DIS
LIN {X -107.7448,Y 61.5372,Z 140,A 146.854,B 23.6871,C -1.4253,E1 23.5883,E2 299.7632} C_DIS
LIN {X -109.0803,Y 59.1381,Z 140,A 148.4554,B 23.6865,C -1.4356,E1 23.586,E2 298.127} C_DIS
LIN {X -110.8834,Y 55.6832,Z 140,A 150.1292,B 23.6871,C -1.425,E1 23.5839,E2 296.4703} C_DIS
LIN {X -112.2351,Y 52.9056,Z 140,A 151.5548,B 23.6874,C -1.4207,E1 23.5822,E2 295.0474} C_DIS
LIN {X -113.7342,Y 49.5983,Z 140,A 153.1109,B 23.6879,C -1.4106,E1 23.5805,E2 293.5076} C_DIS
LIN {X -115.705,Y 44.8072,Z 140,A 155.6661,B 23.6879,C -1.41,E1 23.5778,E2 290.9386} C_DIS
LIN {X -116.8069,Y 41.8512,Z 140,A 157.1648,B 23.6881,C -1.4072,E1 23.5763,E2 289.4378} C_DIS
LIN {X -118.0025,Y 38.3555,Z 140,A 159.0586,B 23.688,C -1.4098,E1 23.5746,E2 287.5262} C_DIS
LIN {X -119.3183,Y 34.0428,Z 140,A 160.9107,B 23.6889,C -1.3935,E1 23.5732,E2 285.7034} C_DIS
LIN {X -119.9479,Y 31.7473,Z 140,A 162.1843,B 23.6887,C -1.3974,E1 23.5723,E2 284.4123} C_DIS
LIN {X -120.7712,Y 28.4615,Z 140,A 163.6265,B 23.6892,C -1.3872,E1 23.5713,E2 282.9866} C_DIS
LIN {X -121.5163,Y 25.0854,Z 140,A 165.6806,B 23.6884,C -1.4014,E1 23.5701,E2 280.8843} C_DIS
LIN {X -122.1899,Y 21.566,Z 140,A 166.9215,B 23.6897,C -1.3786,E1 23.5695,E2 279.6925} C_DIS
LIN {X -122.9087,Y 17.0028,Z 140,A 169.3028,B 23.6895,C -1.3821,E1 23.5685,E2 277.2873} C_DIS
LIN {X -123.8205,Y 8.002,Z 140,A 173.1104,B 23.6911,C -1.353,E1 23.5676,E2 273.5284} C_DIS
LIN {X -124.0766,Y 0.8599,Z 140,A 177.0648,B 23.6902,C -1.3698,E1 23.5673,E2 269.5068} C_DIS
LIN {X -124.0458,Y -2.8922,Z 140,A 178.4584,B 23.6913,C -1.3498,E1 23.5673,E2 268.1541} C_DIS
LIN {X -123.8989,Y -6.6857,Z 140,A -179.9196,B 23.6919,C -1.3387,E1 23.5675,E2 266.5497} C_DIS
LIN {X -123.6545,Y -10.2471,Z 140,A -177.5849,B 23.6906,C -1.3624,E1 23.5681,E2 264.1408} C_DIS
LIN {X -123.1888,Y -14.8298,Z 140,A -176.0431,B 23.6923,C -1.3308,E1 23.5686,E2 262.6682} C_DIS
LIN {X -122.4902,Y -19.7889,Z 140,A -173.3592,B 23.6918,C -1.3392,E1 23.5697,E2 259.9464} C_DIS
LIN {X -121.8983,Y -23.1559,Z 140,A -172.1005,B 23.6928,C -1.3207,E1 23.5703,E2 258.7261} C_DIS
LIN {X -120.8752,Y -28.0123,Z 140,A -169.9198,B 23.6934,C -1.3088,E1 23.5716,E2 256.5615} C_DIS
LIN {X -120.1277,Y -31.0645,Z 140,A -168.4512,B 23.6936,C -1.3051,E1 23.5726,E2 255.0933} C_DIS
LIN {X -119.3184,Y -34.0423,Z 140,A -166.8437,B 23.6934,C -1.3084,E1 23.5738,E2 253.4675} C_DIS
LIN {X -118.2407,Y -37.6095,Z 140,A -165.0926,B 23.6937,C -1.3045,E1 23.5753,E2 251.7155} C_DIS
LIN {X -117.0906,Y -41.0524,Z 140,A -163.5563,B 23.6942,C -1.2935,E1 23.5767,E2 250.1974} C_DIS
LIN {X -116.1661,Y -43.5978,Z 140,A -162.2618,B 23.6943,C -1.2917,E1 23.5779,E2 248.8997} C_DIS
LIN {X -114.9646,Y -46.6749,Z 140,A -160.6601,B 23.6943,C -1.2905,E1 23.5796,E2 247.2916} C_DIS
LIN {X -113.1945,Y -50.8166,Z 140,A -158.7185,B 23.695,C -1.2786,E1 23.5817,E2 245.3683} C_DIS
LIN {X -111.9439,Y -53.515,Z 140,A -157.0062,B 23.6944,C -1.2891,E1 23.5838,E2 243.6197} C_DIS
LIN {X -110.245,Y -56.9372,Z 140,A -155.4966,B 23.6953,C -1.2733,E1 23.5857,E2 242.1412} C_DIS
LIN {X -108.9202,Y -59.432,Z 140,A -154.0746,B 23.6952,C -1.2747,E1 23.5876,E2 240.7076} C_DIS
LIN {X -106.8012,Y -63.1616,Z 140,A -152.036,B 23.6953,C -1.2718,E1 23.5905,E2 238.665} C_DIS
LIN {X -104.5207,Y -66.8669,Z 140,A -150.0573,B 23.6957,C -1.2653,E1 23.5934,E2 236.6921} C_DIS
LIN {X -102.4324,Y -70.0244,Z 140,A -148.2963,B 23.6959,C -1.2613,E1 23.5961,E2 234.9316} C_DIS
LIN {X -100.0206,Y -73.4277,Z 140,A -146.3243,B 23.6959,C -1.2585,E1 23.5994,E2 232.9566} C_DIS
LIN {X -97.2946,Y -77.0042,Z 140,A -144.2415,B 23.6962,C -1.2537,E1 23.6029,E2 230.8752} C_DIS
LIN {X -94.2115,Y -80.7464,Z 140,A -141.3426,B 23.6951,C -1.2772,E1 23.6083,E2 227.9035} C_DIS
LIN {X -90.6457,Y -84.7299,Z 140,A -139.5638,B 23.6968,C -1.2415,E1 23.6115,E2 226.2055} C_DIS
LIN {X -87.7182,Y -87.7577,Z 140,A -137.5632,B 23.6969,C -1.2398,E1 23.6154,E2 224.2003} C_DIS
LIN {X -84.6688,Y -90.7027,Z 140,A -135.6288,B 23.6972,C -1.2347,E1 23.6194,E2 222.2701} C_DIS
LIN {X -81.5453,Y -93.5207,Z 140,A -133.5932,B 23.6972,C -1.2349,E1 23.6236,E2 220.2255} C_DIS
LIN {X -78.7539,Y -95.8837,Z 140,A -131.9277,B 23.6974,C -1.2307,E1 23.6272,E2 218.5638} C_DIS
LIN {X -75.2396,Y -98.665,Z 140,A -129.9007,B 23.6976,C -1.225,E1 23.6317,E2 216.5431} C_DIS
LIN {X -72.149,Y -100.9469,Z 140,A -127.8242,B 23.6971,C -1.2353,E1 23.6364,E2 214.4331} C_DIS
LIN {X -69.2703,Y -102.9442,Z 140,A -126.5995,B 23.6981,C -1.2153,E1 23.6392,E2 213.2541} C_DIS
LIN {X -66.235,Y -104.9222,Z 140,A -124.6535,B 23.6977,C -1.2248,E1 23.6438,E2 211.2778} C_DIS
LIN {X -61.989,Y -107.4856,Z 140,A -122.5008,B 23.6981,C -1.2153,E1 23.649,E2 209.1419} C_DIS
LIN {X -58.2981,Y -109.5313,Z 140,A -120.4479,B 23.6981,C -1.2173,E1 23.654,E2 207.0778} C_DIS
LIN {X -54.6367,Y -111.4011,Z 140,A -118.771,B 23.6986,C -1.2051,E1 23.6581,E2 205.4267} C_DIS
LIN {X -51.8498,Y -112.7252,Z 140,A -117.2815,B 23.6986,C -1.2063,E1 23.6619,E2 203.9302} C_DIS
LIN {X -48.6167,Y -114.1586,Z 140,A -115.4709,B 23.6983,C -1.2124,E1 23.6666,E2 202.0997} C_DIS
LIN {X -44.6388,Y -115.7705,Z 140,A -113.6146,B 23.6986,C -1.2049,E1 23.6714,E2 200.258} C_DIS
LIN {X -41.2681,Y -117.0158,Z 140,A -111.8951,B 23.6986,C -1.2061,E1 23.6759,E2 198.5319} C_DIS
LIN {X -37.0834,Y -118.4088,Z 140,A -110.0309,B 23.699,C -1.1967,E1 23.6808,E2 196.6875} C_DIS
LIN {X -33.8692,Y -119.3668,Z 140,A -108.5852,B 23.6993,C -1.191,E1 23.6847,E2 195.2535} C_DIS
LIN {X -27.2638,Y -121.0462,Z 140,A -105.4529,B 23.6994,C -1.1885,E1 23.6932,E2 192.1227} C_DIS
LIN {X -24.5814,Y -121.6188,Z 140,A -104.0355,B 23.6991,C -1.1947,E1 23.6971,E2 190.688} C_DIS
LIN {X -21.221,Y -122.2516,Z 140,A -102.3164,B 23.6988,C -1.2005,E1 23.7019,E2 188.9526} C_DIS
LIN {X -17.5075,Y -122.8368,Z 140,A -100.6562,B 23.699,C -1.1966,E1 23.7064,E2 187.3007} C_DIS
LIN {X -14.3777,Y -123.2428,Z 140,A -99.2919,B 23.6992,C -1.1921,E1 23.7102,E2 185.9466} C_DIS
LIN {X -11.2209,Y -123.5714,Z 140,A -97.6206,B 23.6988,C -1.2014,E1 23.7149,E2 184.2512} C_DIS
LIN {X -7.419,Y -123.8564,Z 140,A -95.923,B 23.6989,C -1.1985,E1 23.7196,E2 182.5601} C_DIS
LIN {X -3.256,Y -124.0357,Z 140,A -93.9837,B 23.6989,C -1.1995,E1 23.725,E2 180.6182} C_DIS
LIN {X 0.8758,Y -124.0739,Z 140,A -92.875,B 23.7006,C -1.1632,E1 23.7279,E2 179.5997} C_DIS
Enddeposition()
LIN {X 0.8758,Y -124.0739,Z 140,A -92.875,B 23.7006,C -1.1632,E1 23.7279,E2 179.5997} C_DIS
Startdeposition()
$VEL.CP = VEL_PRINT
LIN {X -0.2178,Y -123.1041,Z 140,A -93.0998,B 23.0025,C -1.059,E1 23.0248,E2 179.9955} C_DIS
LIN {X -3.2341,Y -123.061,Z 140,A -94.6766,B 23.0028,C -1.0512,E1 23.0204,E2 181.5923} C_DIS
LIN {X -7.3621,Y -122.8831,Z 140,A -96.654,B 23.0029,C -1.0488,E1 23.0148,E2 183.5766} C_DIS
LIN {X -12.0714,Y -122.5103,Z 140,A -98.6907,B 23.0026,C -1.056,E1 23.0092,E2 185.596} C_DIS
LIN {X -15.0709,Y -122.1782,Z 140,A -100.1091,B 23.0026,C -1.0556,E1 23.0053,E2 187.0164} C_DIS
LIN {X -18.7496,Y -121.6669,Z 140,A -101.8489,B 23.0026,C -1.0556,E1 23.0005,E2 188.7578} C_DIS
LIN {X -21.9062,Y -121.1385,Z 140,A -103.4177,B 23.0028,C -1.0526,E1 22.9961,E2 190.3358} C_DIS
LIN {X -25.4976,Y -120.4345,Z 140,A -105.0938,B 23.0027,C -1.0545,E1 22.9915,E2 192.0092} C_DIS
LIN {X -28.6897,Y -119.7134,Z 140,A -106.5874,B 23.0027,C -1.0566,E1 22.9875,E2 193.4997} C_DIS
LIN {X -32.0865,Y -118.8484,Z 140,A -108.3413,B 23.0027,C -1.0524,E1 22.9827,E2 195.2672} C_DIS
LIN {X -35.7474,Y -117.7988,Z 140,A -109.9996,B 23.0025,C -1.0585,E1 22.9783,E2 196.9129} C_DIS
LIN {X -38.6227,Y -116.8875,Z 140,A -111.3516,B 23.0024,C -1.0618,E1 22.9747,E2 198.259} C_DIS
LIN {X -41.872,Y -115.763,Z 140,A -112.8521,B 23.0021,C -1.0674,E1 22.9708,E2 199.7483} C_DIS
LIN {X -44.4997,Y -114.7785,Z 140,A -114.2034,B 23.0021,C -1.0667,E1 22.9673,E2 201.1045} C_DIS
LIN {X -47.1163,Y -113.7299,Z 140,A -115.5773,B 23.0022,C -1.0654,E1 22.9637,E2 202.4851} C_DIS
LIN {X -50.0841,Y -112.4541,Z 140,A -117.0877,B 23.0022,C -1.0668,E1 22.9598,E2 203.996} C_DIS
LIN {X -52.6351,Y -111.2838,Z 140,A -118.3916,B 23.0021,C -1.0684,E1 22.9565,E2 205.2992} C_DIS
LIN {X -55.548,Y -109.8582,Z 140,A -119.9052,B 23.0021,C -1.0701,E1 22.9527,E2 206.8128} C_DIS
LIN {X -58.223,Y -108.4659,Z 140,A -121.3207,B 23.002,C -1.0714,E1 22.9492,E2 208.2293} C_DIS
LIN {X -60.6777,Y -107.1127,Z 140,A -122.6275,B 23.0019,C -1.0731,E1 22.9461,E2 209.5359} C_DIS
LIN {X -63.5316,Y -105.4445,Z 140,A -124.1485,B 23.0017,C -1.0761,E1 22.9424,E2 211.0543} C_DIS
LIN {X -65.8662,Y -104.0021,Z 140,A -125.5946,B 23.002,C -1.071,E1 22.9389,E2 212.5184} C_DIS
LIN {X -69.489,Y -101.6173,Z 140,A -127.524,B 23.0017,C -1.078,E1 22.9345,E2 214.437} C_DIS
LIN {X -72.1212,Y -99.7663,Z 140,A -128.9775,B 23.0015,C -1.0824,E1 22.9312,E2 215.8847} C_DIS
LIN {X -75.0852,Y -97.5557,Z 140,A -130.8707,B 23.0017,C -1.0783,E1 22.9269,E2 217.7959} C_DIS
LIN {X -78.0945,Y -95.1634,Z 140,A -132.6698,B 23.0015,C -1.0812,E1 22.923,E2 219.595} C_DIS
LIN {X -81.6423,Y -92.1375,Z 140,A -134.6881,B 23.0011,C -1.0917,E1 22.9188,E2 221.5949} C_DIS
LIN {X -84.3439,Y -89.6711,Z 140,A -136.5233,B 23.0011,C -1.0897,E1 22.915,E2 223.4434} C_DIS
LIN {X -87.5079,Y -86.5863,Z 140,A -138.5867,B 23.001,C -1.0938,E1 22.9109,E2 225.5059} C_DIS
LIN {X -90.3827,Y -83.5815,Z 140,A -140.5404,B 23.0008,C -1.0973,E1 22.9072,E2 227.4599} C_DIS
LIN {X -93.2383,Y -80.3827,Z 140,A -142.4077,B 23.0004,C -1.1071,E1 22.9038,E2 229.3113} C_DIS
LIN {X -95.2354,Y -78.0064,Z 140,A -143.9945,B 23.0004,C -1.1047,E1 22.9009,E2 230.9123} C_DIS
LIN {X -97.9738,Y -74.5385,Z 140,A -145.9792,B 23.0001,C -1.1126,E1 22.8975,E2 232.8871} C_DIS
LIN {X -100.3456,Y -71.3138,Z 140,A -147.9747,B 23.0001,C -1.1118,E1 22.8943,E2 234.8951} C_DIS
LIN {X -102.4757,Y -68.2166,Z 140,A -149.5724,B 22.9997,C -1.1224,E1 22.8918,E2 236.4742} C_DIS
LIN {X -104.1122,Y -65.6919,Z 140,A -151.1061,B 22.9997,C -1.1207,E1 22.8895,E2 238.021} C_DIS
LIN {X -106.3715,Y -61.9675,Z 140,A -153.0128,B 22.9993,C -1.1309,E1 22.8868,E2 239.9121} C_DIS
LIN {X -107.8518,Y -59.3536,Z 140,A -154.4306,B 22.9991,C -1.1339,E1 22.8848,E2 241.3304} C_DIS
LIN {X -109.273,Y -56.6929,Z 140,A -155.8628,B 22.999,C -1.1367,E1 22.883,E2 242.7638} C_DIS
LIN {X -110.7292,Y -53.7949,Z 140,A -157.5073,B 22.999,C -1.1355,E1 22.8809,E2 244.4212} C_DIS
LIN {X -112.4533,Y -50.0859,Z 140,A -159.3314,B 22.9986,C -1.1441,E1 22.8788,E2 246.2341} C_DIS
LIN {X -114.0708,Y -46.2843,Z 140,A -161.2545,B 22.9984,C -1.1496,E1 22.8767,E2 248.1546} C_DIS
LIN {X -115.3914,Y -42.8865,Z 140,A -162.9433,B 22.9981,C -1.1549,E1 22.8751,E2 249.8402} C_DIS
LIN {X -116.4773,Y -39.8451,Z 140,A -164.4155,B 22.9979,C -1.1606,E1 22.8737,E2 251.3069} C_DIS
LIN {X -117.5751,Y -36.4783,Z 140,A -165.9736,B 22.9975,C -1.1691,E1 22.8724,E2 252.8528} C_DIS
LIN {X -118.2947,Y -34.0735,Z 140,A -167.266,B 22.9975,C -1.1677,E1 22.8714,E2 254.1572} C_DIS
LIN {X -119.0391,Y -31.3715,Z 140,A -168.5794,B 22.9973,C -1.1714,E1 22.8704,E2 255.4696} C_DIS
LIN {X -119.7721,Y -28.4458,Z 140,A -170.0096,B 22.9972,C -1.1746,E1 22.8695,E2 256.9005} C_DIS
LIN {X -120.4816,Y -25.2795,Z 140,A -171.5065,B 22.9969,C -1.1798,E1 22.8686,E2 258.3938} C_DIS
LIN {X -121.058,Y -22.3563,Z 140,A -172.8971,B 22.9967,C -1.184,E1 22.8679,E2 259.7826} C_DIS
LIN {X -121.5514,Y -19.4962,Z 140,A -174.2747,B 22.9966,C -1.1872,E1 22.8672,E2 261.161} C_DIS
LIN {X -122.0111,Y -16.3654,Z 140,A -175.6867,B 22.9962,C -1.1942,E1 22.8667,E2 262.564} C_DIS
LIN {X -122.3687,Y -13.4302,Z 140,A -177.2474,B 22.9964,C -1.1913,E1 22.8662,E2 264.1426} C_DIS
LIN {X -122.7543,Y -9.2674,Z 140,A -179.1987,B 22.9961,C -1.1973,E1 22.8657,E2 266.0914} C_DIS
LIN {X -122.9654,Y -5.8355,Z 140,A 179.3121,B 22.9956,C -1.2068,E1 22.8655,E2 267.5658} C_DIS
LIN {X -123.0798,Y -2.4389,Z 140,A 177.6567,B 22.9956,C -1.2089,E1 22.8653,E2 269.2266} C_DIS
LIN {X -123.1008,Y 0.9666,Z 140,A 175.8933,B 22.9956,C -1.207,E1 22.8653,E2 271.0069} C_DIS
LIN {X -123.019,Y 4.5612,Z 140,A 174.4026,B 22.995,C -1.2196,E1 22.8655,E2 272.4748} C_DIS
LIN {X -122.8319,Y 8.1935,Z 140,A 172.7307,B 22.9947,C -1.2258,E1 22.8657,E2 274.1417} C_DIS
LIN {X -122.647,Y 10.5908,Z 140,A 171.5814,B 22.9945,C -1.2283,E1 22.866,E2 275.2922} C_DIS
LIN {X -122.3307,Y 13.7835,Z 140,A 170.0893,B 22.9943,C -1.2331,E1 22.8664,E2 276.7817} C_DIS
LIN {X -121.9525,Y 16.8033,Z 140,A 168.6323,B 22.9941,C -1.236,E1 22.867,E2 278.2407} C_DIS
LIN {X -121.5061,Y 19.771,Z 140,A 167.168,B 22.9941,C -1.2379,E1 22.8676,E2 279.7099} C_DIS
LIN {X -120.9818,Y 22.7579,Z 140,A 165.8807,B 22.9936,C -1.2473,E1 22.8682,E2 280.9813} C_DIS
LIN {X -120.4327,Y 25.5059,Z 140,A 164.4311,B 22.9936,C -1.2457,E1 22.8691,E2 282.4445} C_DIS
LIN {X -119.7218,Y 28.6545,Z 140,A 162.9828,B 22.9933,C -1.2526,E1 22.87,E2 283.8843} C_DIS
LIN {X -118.9327,Y 31.7704,Z 140,A 161.5844,B 22.9929,C -1.2612,E1 22.8709,E2 285.2694} C_DIS
LIN {X -118.2331,Y 34.2837,Z 140,A 160.2531,B 22.9929,C -1.2604,E1 22.872,E2 286.6113} C_DIS
LIN {X -117.2934,Y 37.3711,Z 140,A 158.7988,B 22.9926,C -1.267,E1 22.8732,E2 288.0578} C_DIS
LIN {X -116.4076,Y 40.0461,Z 140,A 157.2963,B 22.9927,C -1.2635,E1 22.8745,E2 289.5788} C_DIS
LIN {X -115.3728,Y 42.936,Z 140,A 155.9298,B 22.9924,C -1.2703,E1 22.8758,E2 290.9361} C_DIS
LIN {X -114.0555,Y 46.3223,Z 140,A 154.1658,B 22.9923,C -1.2726,E1 22.8777,E2 292.7051} C_DIS
LIN {X -112.4516,Y 50.0896,Z 140,A 152.3612,B 22.9917,C -1.2824,E1 22.8796,E2 294.4954} C_DIS
LIN {X -111.2825,Y 52.6377,Z 140,A 150.9874,B 22.9917,C -1.2835,E1 22.8813,E2 295.8745} C_DIS
LIN {X -109.8647,Y 55.5352,Z 140,A 149.5337,B 22.9913,C -1.2899,E1 22.8831,E2 297.3204} C_DIS
LIN {X -108.4742,Y 58.2075,Z 140,A 148.1247,B 22.9911,C -1.2937,E1 22.8849,E2 298.7279} C_DIS
LIN {X -107.1214,Y 60.6623,Z 140,A 146.804,B 22.991,C -1.2968,E1 22.8867,E2 300.0482} C_DIS
LIN {X -105.3938,Y 63.6154,Z 140,A 145.0659,B 22.991,C -1.2956,E1 22.8892,E2 301.7993} C_DIS
LIN {X -103.1837,Y 67.1408,Z 140,A 143.254,B 22.9905,C -1.306,E1 22.8919,E2 303.5945} C_DIS
LIN {X -101.3863,Y 69.8256,Z 140,A 141.7828,B 22.9902,C -1.3114,E1 22.8942,E2 305.0596} C_DIS
LIN {X -99.7691,Y 72.1173,Z 140,A 140.4334,B 22.9901,C -1.3132,E1 22.8964,E2 306.4116} C_DIS
LIN {X -97.5783,Y 75.0556,Z 140,A 138.5657,B 22.9902,C -1.3113,E1 22.8996,E2 308.2941} C_DIS
LIN {X -95.1564,Y 78.103,Z 140,A 136.727,B 22.99,C -1.315,E1 22.9028,E2 310.1328} C_DIS
LIN {X -92.222,Y 81.5467,Z 140,A 134.6135,B 22.9897,C -1.32,E1 22.9066,E2 312.2438} C_DIS
LIN {X -89.2331,Y 84.8076,Z 140,A 132.5391,B 22.9895,C -1.3245,E1 22.9106,E2 314.3166} C_DIS
LIN {X -86.2651,Y 87.8242,Z 140,A 130.622,B 22.9891,C -1.3313,E1 22.9144,E2 316.2251} C_DIS
LIN {X -83.2302,Y 90.7056,Z 140,A 128.602,B 22.9891,C -1.3329,E1 22.9185,E2 318.25} C_DIS
LIN {X -80.1149,Y 93.4689,Z 140,A 126.7039,B 22.9887,C -1.3389,E1 22.9225,E2 320.1409} C_DIS
LIN {X -76.9146,Y 96.1197,Z 140,A 124.7136,B 22.9886,C -1.3408,E1 22.9268,E2 322.1345} C_DIS
LIN {X -74.3706,Y 98.1012,Z 140,A 123.3684,B 22.9881,C -1.3503,E1 22.9297,E2 323.4608} C_DIS
LIN {X -71.947,Y 99.8925,Z 140,A 121.9755,B 22.9879,C -1.3535,E1 22.9329,E2 324.8507} C_DIS
LIN {X -69.0625,Y 101.9075,Z 140,A 120.1893,B 22.988,C -1.3507,E1 22.937,E2 326.6507} C_DIS
LIN {X -65.8107,Y 104.0372,Z 140,A 118.4951,B 22.9876,C -1.3588,E1 22.9409,E2 328.3301} C_DIS
LIN {X -63.0733,Y 105.7191,Z 140,A 116.9916,B 22.9875,C -1.3612,E1 22.9445,E2 329.8326} C_DIS
LIN {X -60.6606,Y 107.1224,Z 140,A 115.679,B 22.9874,C -1.3629,E1 22.9477,E2 331.145} C_DIS
LIN {X -58.0266,Y 108.5714,Z 140,A 114.255,B 22.9873,C -1.3643,E1 22.9512,E2 332.57} C_DIS
LIN {X -55.1704,Y 110.0505,Z 140,A 112.7679,B 22.9871,C -1.3671,E1 22.9549,E2 334.0543} C_DIS
LIN {X -52.6254,Y 111.2884,Z 140,A 111.4499,B 22.9871,C -1.3691,E1 22.9582,E2 335.3707} C_DIS
LIN {X -49.6861,Y 112.6322,Z 140,A 109.9402,B 22.9869,C -1.3711,E1 22.9621,E2 336.8793} C_DIS
LIN {X -46.9115,Y 113.8154,Z 140,A 108.3479,B 22.9872,C -1.3653,E1 22.9662,E2 338.4905} C_DIS
LIN {X -42.8876,Y 115.3909,Z 140,A 106.4928,B 22.9867,C -1.3744,E1 22.971,E2 340.3266} C_DIS
LIN {X -39.8277,Y 116.4833,Z 140,A 105.0032,B 22.9866,C -1.3772,E1 22.9749,E2 341.8121} C_DIS
LIN {X -36.9671,Y 117.4225,Z 140,A 103.5989,B 22.9865,C -1.3787,E1 22.9786,E2 343.2153} C_DIS
LIN {X -33.8378,Y 118.3632,Z 140,A 102.092,B 22.9863,C -1.3809,E1 22.9827,E2 344.7194} C_DIS
LIN {X -31.3811,Y 119.0365,Z 140,A 100.8877,B 22.9863,C -1.3813,E1 22.9859,E2 345.9246} C_DIS
LIN {X -28.4586,Y 119.769,Z 140,A 99.3401,B 22.9866,C -1.3766,E1 22.9902,E2 347.4867} C_DIS
LIN {X -25.2846,Y 120.4805,Z 140,A 97.9734,B 22.9862,C -1.384,E1 22.9938,E2 348.8362} C_DIS
LIN {X -21.933,Y 121.1337,Z 140,A 96.5695,B 22.9857,C -1.3931,E1 22.9976,E2 350.2185} C_DIS
LIN {X -19.5444,Y 121.5439,Z 140,A 95.2277,B 22.9861,C -1.3848,E1 23.0014,E2 351.583} C_DIS
LIN {X -16.3518,Y 122.0129,Z 140,A 93.7301,B 22.9861,C -1.3859,E1 23.0055,E2 353.0789} C_DIS
LIN {X -13.3554,Y 122.3767,Z 140,A 92.3264,B 22.9861,C -1.3868,E1 23.0094,E2 354.4815} C_DIS
LIN {X -9.5626,Y 122.7328,Z 140,A 90.4242,B 22.9863,C -1.3821,E1 23.0147,E2 356.3967} C_DIS
LIN {X -5.8182,Y 122.9663,Z 140,A 88.8432,B 22.9858,C -1.3897,E1 23.0191,E2 357.9587} C_DIS
LIN {X -2.8049,Y 123.0729,Z 140,A 87.4337,B 22.9858,C -1.3898,E1 23.023,E2 359.3681} C_DIS
LIN {X 0.2134,Y 123.1041,Z 140,A 86.0523,B 22.9858,C -1.3911,E1 23.0269,E2 360.7462} C_DIS
LIN {X 3.3654,Y 123.0573,Z 140,A 84.476,B 22.986,C -1.3866,E1 23.0313,E2 362.3337} C_DIS
LIN {X 7.3457,Y 122.8841,Z 140,A 82.5908,B 22.986,C -1.3853,E1 23.0366,E2 364.2215} C_DIS
LIN {X 10.5643,Y 122.6493,Z 140,A 81.1796,B 22.9859,C -1.3891,E1 23.0405,E2 365.6223} C_DIS
LIN {X 13.7792,Y 122.3311,Z 140,A 79.5275,B 22.9863,C -1.3824,E1 23.0451,E2 367.2902} C_DIS
LIN {X 17.6066,Y 121.8377,Z 140,A 77.8247,B 22.9861,C -1.386,E1 23.0498,E2 368.9822} C_DIS
LIN {X 21.2595,Y 121.2543,Z 140,A 76.0263,B 22.9863,C -1.3821,E1 23.0548,E2 370.7886} C_DIS
LIN {X 25.3314,Y 120.4704,Z 140,A 74.0999,B 22.9863,C -1.3813,E1 23.06,E2 372.7144} C_DIS
LIN {X 28.8985,Y 119.663,Z 140,A 72.5779,B 22.9859,C -1.3882,E1 23.0641,E2 374.2164} C_DIS
LIN {X 31.3909,Y 119.0339,Z 140,A 71.3299,B 22.9861,C -1.3852,E1 23.0675,E2 375.47} C_DIS
LIN {X 34.2969,Y 118.2293,Z 140,A 69.9295,B 22.9861,C -1.3844,E1 23.0713,E2 376.87} C_DIS
LIN {X 37.3849,Y 117.289,Z 140,A 68.4113,B 22.9863,C -1.3825,E1 23.0753,E2 378.39} C_DIS
LIN {X 40.0478,Y 116.407,Z 140,A 67.074,B 22.9863,C -1.38,E1 23.0789,E2 379.7308} C_DIS
LIN {X 43.6709,Y 115.0976,Z 140,A 65.1787,B 22.9867,C -1.3738,E1 23.0839,E2 381.6376} C_DIS
LIN {X 47.1137,Y 113.731,Z 140,A 63.5446,B 22.9867,C -1.376,E1 23.0881,E2 383.262} C_DIS
LIN {X 50.083,Y 112.4546,Z 140,A 62.1201,B 22.9865,C -1.3778,E1 23.0917,E2 384.6781} C_DIS
LIN {X 52.7376,Y 111.2348,Z 140,A 60.8023,B 22.9865,C -1.378,E1 23.095,E2 385.9916} C_DIS
LIN {X 55.5428,Y 109.8608,Z 140,A 59.2909,B 22.9868,C -1.3736,E1 23.0988,E2 387.5098} C_DIS
LIN {X 58.2159,Y 108.4697,Z 140,A 57.9164,B 22.9868,C -1.3729,E1 23.1022,E2 388.8818} C_DIS
LIN {X 60.688,Y 107.1067,Z 140,A 56.6066,B 22.9868,C -1.3712,E1 23.1054,E2 390.1916} C_DIS
LIN {X 63.4754,Y 105.4784,Z 140,A 54.9751,B 22.9873,C -1.3633,E1 23.1094,E2 391.8379} C_DIS
LIN {X 67.5275,Y 102.9313,Z 140,A 52.7403,B 22.9876,C -1.3594,E1 23.1146,E2 394.0746} C_DIS
LIN {X 70.8889,Y 100.6456,Z 140,A 51.0058,B 22.9873,C -1.3633,E1 23.1186,E2 395.7927} C_DIS
LIN {X 73.3335,Y 98.8788,Z 140,A 49.4541,B 22.9878,C -1.3542,E1 23.1221,E2 397.3616} C_DIS
LIN {X 76.9171,Y 96.1178,Z 140,A 47.3426,B 22.9881,C -1.35,E1 23.1267,E2 399.4751} C_DIS
LIN {X 80.3319,Y 93.2821,Z 140,A 45.4082,B 22.988,C -1.352,E1 23.1308,E2 401.3964} C_DIS
LIN {X 83.2358,Y 90.7004,Z 140,A 43.4979,B 22.9884,C -1.3437,E1 23.1348,E2 403.3193} C_DIS
LIN {X 86.4378,Y 87.6548,Z 140,A 41.5598,B 22.9884,C -1.3447,E1 23.1387,E2 405.2459} C_DIS
LIN {X 89.2296,Y 84.8112,Z 140,A 39.6135,B 22.9888,C -1.3365,E1 23.1425,E2 407.2039} C_DIS
LIN {X 92.2004,Y 81.5712,Z 140,A 37.6049,B 22.989,C -1.3336,E1 23.1462,E2 409.2102} C_DIS
LIN {X 94.7539,Y 78.5904,Z 140,A 35.7811,B 22.9892,C -1.3295,E1 23.1495,E2 411.0354} C_DIS
LIN {X 97.5136,Y 75.1397,Z 140,A 33.806,B 22.9892,C -1.3282,E1 23.1529,E2 413.0036} C_DIS
LIN {X 99.8746,Y 71.9718,Z 140,A 31.8612,B 22.9898,C -1.3188,E1 23.1562,E2 414.9621} C_DIS
LIN {X 102.4775,Y 68.214,Z 140,A 29.9155,B 22.9896,C -1.3217,E1 23.1592,E2 416.8899} C_DIS
LIN {X 104.3721,Y 65.2787,Z 140,A 28.1705,B 22.9902,C -1.312,E1 23.1618,E2 418.65} C_DIS
LIN {X 106.6722,Y 61.4482,Z 140,A 26.3791,B 22.9897,C -1.3196,E1 23.1643,E2 420.4118} C_DIS
LIN {X 107.8495,Y 59.3578,Z 140,A 25.121,B 22.9903,C -1.3101,E1 23.1661,E2 421.6869} C_DIS
LIN {X 109.2695,Y 56.6994,Z 140,A 23.7145,B 22.9905,C -1.3061,E1 23.1679,E2 423.0956} C_DIS
LIN {X 110.9085,Y 53.4206,Z 140,A 22.1864,B 22.9903,C -1.3095,E1 23.1698,E2 424.606} C_DIS
LIN {X 111.9225,Y 51.2626,Z 140,A 20.7852,B 22.9912,C -1.2929,E1 23.1715,E2 426.0411} C_DIS
LIN {X 113.4814,Y 47.7114,Z 140,A 19.3317,B 22.9906,C -1.3039,E1 23.173,E2 427.4577} C_DIS
LIN {X 114.5452,Y 45.0999,Z 140,A 17.9284,B 22.991,C -1.2959,E1 23.1745,E2 428.873} C_DIS
LIN {X 115.3899,Y 42.8903,Z 140,A 16.7189,B 22.9915,C -1.2876,E1 23.1757,E2 430.0962} C_DIS
LIN {X 116.5168,Y 39.731,Z 140,A 15.2034,B 22.9916,C -1.2851,E1 23.1771,E2 431.6088} C_DIS
LIN {X 117.438,Y 36.9184,Z 140,A 13.8263,B 22.9918,C -1.2809,E1 23.1783,E2 432.9879} C_DIS
LIN {X 118.2993,Y 34.0577,Z 140,A 12.4466,B 22.992,C -1.2772,E1 23.1794,E2 434.3684} C_DIS
LIN {X 119.2722,Y 30.4717,Z 140,A 10.5386,B 22.9927,C -1.2637,E1 23.1807,E2 436.2988} C_DIS
LIN {X 120.1607,Y 26.762,Z 140,A 8.8013,B 22.9929,C -1.2599,E1 23.1818,E2 438.0347} C_DIS
LIN {X 120.9849,Y 22.7414,Z 140,A 7.0561,B 22.9929,C -1.2616,E1 23.1828,E2 439.7644} C_DIS
LIN {X 121.6071,Y 19.1362,Z 140,A 5.3212,B 22.9932,C -1.2548,E1 23.1836,E2 441.5055} C_DIS
LIN {X 122.0129,Y 16.3518,Z 140,A 4.1377,B 22.9931,C -1.2565,E1 23.184,E2 442.6769} C_DIS
LIN {X 122.3766,Y 13.357,Z 140,A 2.679,B 22.9935,C -1.2495,E1 23.1845,E2 444.144} C_DIS
LIN {X 122.6493,Y 10.5637,Z 140,A 1.2619,B 22.9939,C -1.2402,E1 23.1848,E2 445.5757} C_DIS
LIN {X 122.9482,Y 6.177,Z 140,A -0.6945,B 22.9941,C -1.2378,E1 23.1852,E2 447.5253} C_DIS
LIN {X 123.0728,Y 2.8074,Z 140,A -2.3043,B 22.9944,C -1.2308,E1 23.1853,E2 449.1423} C_DIS
LIN {X 123.0953,Y -1.5088,Z 140,A -4.2735,B 22.9946,C -1.2262,E1 23.1853,E2 451.1104} C_DIS
LIN {X 123.0069,Y -4.871,Z 140,A -5.7945,B 22.9948,C -1.2233,E1 23.1852,E2 452.629} C_DIS
LIN {X 122.8489,Y -7.9178,Z 140,A -7.1351,B 22.9948,C -1.2224,E1 23.1849,E2 453.9631} C_DIS
LIN {X 122.6494,Y -10.5634,Z 140,A -8.5401,B 22.9954,C -1.2105,E1 23.1846,E2 455.3893} C_DIS
LIN {X 122.3313,Y -13.7773,Z 140,A -9.8582,B 22.9952,C -1.2142,E1 23.1842,E2 456.6892} C_DIS
LIN {X 121.9573,Y -16.77,Z 140,A -11.4129,B 22.9958,C -1.2027,E1 23.1837,E2 458.2633} C_DIS
LIN {X 121.4054,Y -20.3745,Z 140,A -12.954,B 22.9958,C -1.2045,E1 23.183,E2 459.7898} C_DIS
LIN {X 120.7304,Y -24.0581,Z 140,A -14.6917,B 22.996,C -1.1992,E1 23.1821,E2 461.53} C_DIS
LIN {X 120.0605,Y -27.2007,Z 140,A -16.1739,B 22.9962,C -1.195,E1 23.1812,E2 463.0133} C_DIS
LIN {X 119.3605,Y -30.124,Z 140,A -17.5918,B 22.9965,C -1.1897,E1 23.1802,E2 464.4357} C_DIS
LIN {X 118.6453,Y -32.829,Z 140,A -18.8609,B 22.9965,C -1.1871,E1 23.1793,E2 465.7033} C_DIS
LIN {X 117.8011,Y -35.7398,Z 140,A -20.3093,B 22.9969,C -1.1809,E1 23.1782,E2 467.1585} C_DIS
LIN {X 116.8904,Y -38.6143,Z 140,A -21.6513,B 22.9969,C -1.1794,E1 23.177,E2 468.496} C_DIS
LIN {X 115.8342,Y -41.6746,Z 140,A -23.1895,B 22.9973,C -1.1733,E1 23.1756,E2 470.0404} C_DIS
LIN {X 114.7781,Y -44.5007,Z 140,A -24.4792,B 22.9973,C -1.1743,E1 23.1743,E2 471.3196} C_DIS
LIN {X 113.6676,Y -47.2654,Z 140,A -25.8626,B 22.9974,C -1.1702,E1 23.1729,E2 472.705} C_DIS
LIN {X 112.46,Y -50.0709,Z 140,A -27.326,B 22.9977,C -1.1639,E1 23.1712,E2 474.1756} C_DIS
LIN {X 111.2895,Y -52.6232,Z 140,A -28.6198,B 22.9979,C -1.1606,E1 23.1697,E2 475.4703} C_DIS
LIN {X 109.8568,Y -55.5508,Z 140,A -30.1281,B 22.9981,C -1.1565,E1 23.1678,E2 476.9801} C_DIS
LIN {X 108.4629,Y -58.2286,Z 140,A -31.5269,B 22.9982,C -1.1526,E1 23.166,E2 478.3807} C_DIS
LIN {X 107.1097,Y -60.6828,Z 140,A -32.8238,B 22.9984,C -1.1491,E1 23.1642,E2 479.679} C_DIS
LIN {X 105.4806,Y -63.4719,Z 140,A -34.4574,B 22.9989,C -1.1388,E1 23.1619,E2 481.3298} C_DIS
LIN {X 103.1818,Y -67.1439,Z 140,A -36.3223,B 22.9989,C -1.1401,E1 23.1591,E2 483.181} C_DIS
LIN {X 101.3863,Y -69.8256,Z 140,A -37.7741,B 22.9989,C -1.1382,E1 23.1568,E2 484.6297} C_DIS
LIN {X 99.7699,Y -72.1163,Z 140,A -39.1055,B 22.9991,C -1.1334,E1 23.1546,E2 485.9662} C_DIS
LIN {X 97.556,Y -75.0848,Z 140,A -40.9853,B 22.9997,C -1.1215,E1 23.1514,E2 487.8665} C_DIS
LIN {X 95.1505,Y -78.1103,Z 140,A -42.7718,B 22.9999,C -1.1174,E1 23.1483,E2 489.6544} C_DIS
LIN {X 92.2896,Y -81.4702,Z 140,A -44.6969,B 22.9999,C -1.118,E1 23.1448,E2 491.5684} C_DIS
LIN {X 89.6549,Y -84.3611,Z 140,A -46.5845,B 23.0002,C -1.1104,E1 23.1412,E2 493.4664} C_DIS
LIN {X 86.5756,Y -87.5186,Z 140,A -48.5375,B 23.0002,C -1.1099,E1 23.1374,E2 495.4114} C_DIS
LIN {X 83.7049,Y -90.268,Z 140,A -50.4851,B 23.0006,C -1.1011,E1 23.1334,E2 497.3727} C_DIS
LIN {X 80.8826,Y -92.805,Z 140,A -52.2579,B 23.0008,C -1.0967,E1 23.1297,E2 499.1488} C_DIS
LIN {X 77.5028,Y -95.646,Z 140,A -54.2957,B 23.001,C -1.093,E1 23.1253,E2 501.1877} C_DIS
LIN {X 74.3706,Y -98.1012,Z 140,A -55.9819,B 23.0008,C -1.0966,E1 23.1216,E2 502.8579} C_DIS
LIN {X 71.9467,Y -99.8928,Z 140,A -57.3617,B 23.0009,C -1.0947,E1 23.1185,E2 504.2371} C_DIS
LIN {X 69.4601,Y -101.6371,Z 140,A -58.7966,B 23.0011,C -1.0909,E1 23.1152,E2 505.6763} C_DIS
LIN {X 66.9475,Y -103.3093,Z 140,A -60.1427,B 23.0011,C -1.0909,E1 23.1121,E2 507.0177} C_DIS
LIN {X 64.5216,Y -104.8416,Z 140,A -61.5543,B 23.0014,C -1.0849,E1 23.1087,E2 508.4396} C_DIS
LIN {X 61.8046,Y -106.4659,Z 140,A -62.9254,B 23.0013,C -1.0868,E1 23.1054,E2 509.8011} C_DIS
LIN {X 59.3623,Y -107.847,Z 140,A -64.2924,B 23.0015,C -1.0818,E1 23.1021,E2 511.1766} C_DIS
LIN {X 56.7012,Y -109.2686,Z 140,A -65.8509,B 23.0019,C -1.0724,E1 23.0982,E2 512.7541} C_DIS
LIN {X 53.4585,Y -110.8904,Z 140,A -67.235,B 23.0014,C -1.0834,E1 23.0948,E2 514.1061} C_DIS
LIN {X 51.2523,Y -111.9273,Z 140,A -68.5192,B 23.0018,C -1.0749,E1 23.0915,E2 515.4085} C_DIS
LIN {X 48.2993,Y -113.2336,Z 140,A -70.0118,B 23.0018,C -1.0731,E1 23.0877,E2 516.9017} C_DIS
LIN {X 44.5005,Y -114.7782,Z 140,A -71.9354,B 23.002,C -1.0698,E1 23.0827,E2 518.829} C_DIS
LIN {X 41.2615,Y -115.9831,Z 140,A -73.5033,B 23.002,C -1.0695,E1 23.0786,E2 520.394} C_DIS
LIN {X 38.5296,Y -116.9186,Z 140,A -74.8608,B 23.0021,C -1.0673,E1 23.075,E2 521.7544} C_DIS
LIN {X 35.4838,Y -117.8794,Z 140,A -76.3227,B 23.0021,C -1.0666,E1 23.0711,E2 523.215} C_DIS
LIN {X 32.6166,Y -118.7048,Z 140,A -77.6943,B 23.0021,C -1.0659,E1 23.0674,E2 524.5861} C_DIS
LIN {X 29.208,Y -119.5884,Z 140,A -79.5054,B 23.0026,C -1.0566,E1 23.0624,E2 526.4178} C_DIS
LIN {X 25.2802,Y -120.4815,Z 140,A -81.2062,B 23.0023,C -1.0626,E1 23.0578,E2 528.1009} C_DIS
LIN {X 22.5292,Y -121.0255,Z 140,A -82.5096,B 23.0023,C -1.0616,E1 23.0542,E2 529.4051} C_DIS
LIN {X 19.0114,Y -121.6264,Z 140,A -84.2223,B 23.0025,C -1.0581,E1 23.0495,E2 531.1248} C_DIS
LIN {X 16.3464,Y -122.0136,Z 140,A -85.3672,B 23.0024,C -1.0621,E1 23.0464,E2 532.2585} C_DIS
LIN {X 13.352,Y -122.3771,Z 140,A -86.8678,B 23.0026,C -1.057,E1 23.0422,E2 533.7709} C_DIS
LIN {X 10.5595,Y -122.6497,Z 140,A -88.1399,B 23.0026,C -1.0578,E1 23.0386,E2 535.04} C_DIS
LIN {X 6.7913,Y -122.9174,Z 140,A -90.0795,B 23.0029,C -1.0491,E1 23.0332,E2 537.001} C_DIS
LIN {X 2.3459,Y -123.0814,Z 140,A -91.7707,B 23.0022,C -1.0651,E1 23.0286,E2 538.6509} C_DIS
LIN {X 2.3459,Y -123.0814,Z 140,A -91.7707,B 23.0022,C -1.0651,E1 23.0286,E2 538.6509} C_DIS
Enddeposition()
LIN {X 0.9099,Y -128.3847,Z 141,A -92.8842,B 24.9657,C -1.3524,E1 25.0012,E2 539.3203} C_DIS
Startdeposition()
$VEL.CP = VEL_PRINT
LIN {X -3.7539,Y -128.3329,Z 141,A -95.1648,B 24.9663,C -1.342,E1 24.9948,E2 541.6255} C_DIS
LIN {X -6.7791,Y -128.209,Z 141,A -96.5597,B 24.9663,C -1.3397,E1 24.9909,E2 543.0261} C_DIS
LIN {X -11.0309,Y -127.913,Z 141,A -98.4844,B 24.9664,C -1.3386,E1 24.9855,E2 544.9542} C_DIS
LIN {X -15.0345,Y -127.5043,Z 141,A -100.2842,B 24.9664,C -1.3386,E1 24.9805,E2 546.755} C_DIS
LIN {X -18.503,Y -127.0477,Z 141,A -101.7643,B 24.9662,C -1.343,E1 24.9764,E2 548.226} C_DIS
LIN {X -21.4719,Y -126.5797,Z 141,A -103.1758,B 24.9664,C -1.3399,E1 24.9725,E2 549.646} C_DIS
LIN {X -24.8536,Y -125.9612,Z 141,A -104.6787,B 24.9663,C -1.342,E1 24.9684,E2 551.1456} C_DIS
LIN {X -28.934,Y -125.0851,Z 141,A -106.5253,B 24.9662,C -1.3438,E1 24.9634,E2 552.9904} C_DIS
LIN {X -31.9038,Y -124.3607,Z 141,A -107.9287,B 24.9662,C -1.3426,E1 24.9596,E2 554.3985} C_DIS
LIN {X -34.7036,Y -123.6082,Z 141,A -109.2441,B 24.9662,C -1.3424,E1 24.956,E2 555.7165} C_DIS
LIN {X -37.9171,Y -122.661,Z 141,A -110.7473,B 24.9662,C -1.3431,E1 24.952,E2 557.2206} C_DIS
LIN {X -40.9063,Y -121.6968,Z 141,A -112.1534,B 24.9662,C -1.344,E1 24.9483,E2 558.6271} C_DIS
LIN {X -44.2898,Y -120.5086,Z 141,A -113.7224,B 24.966,C -1.3469,E1 24.9441,E2 560.1923} C_DIS
LIN {X -48.3169,Y -118.949,Z 141,A -115.6578,B 24.966,C -1.3485,E1 24.9391,E2 562.1282} C_DIS
LIN {X -51.558,Y -117.5818,Z 141,A -117.2187,B 24.9658,C -1.3506,E1 24.9351,E2 563.6877} C_DIS
LIN {X -54.2219,Y -116.3761,Z 141,A -118.5408,B 24.9658,C -1.3513,E1 24.9317,E2 565.0114} C_DIS
LIN {X -57.1292,Y -114.9768,Z 141,A -119.9864,B 24.9658,C -1.3528,E1 24.9281,E2 566.4572} C_DIS
LIN {X -60.4068,Y -113.2914,Z 141,A -121.7753,B 24.966,C -1.348,E1 24.9237,E2 568.2624} C_DIS
LIN {X -64.0988,Y -111.2437,Z 141,A -123.6534,B 24.9658,C -1.351,E1 24.9191,E2 570.139} C_DIS
LIN {X -68.0607,Y -108.8649,Z 141,A -125.6862,B 24.9656,C -1.3555,E1 24.9143,E2 572.1672} C_DIS
LIN {X -71.6274,Y -106.5525,Z 141,A -127.6354,B 24.9656,C -1.3561,E1 24.9097,E2 574.1215} C_DIS
LIN {X -75.2127,Y -104.052,Z 141,A -129.5645,B 24.9653,C -1.3605,E1 24.9053,E2 576.0468} C_DIS
LIN {X -78.7537,Y -101.3983,Z 141,A -131.4862,B 24.965,C -1.3666,E1 24.9011,E2 577.961} C_DIS
LIN {X -82.0319,Y -98.7651,Z 141,A -133.3601,B 24.9648,C -1.3703,E1 24.897,E2 579.8331} C_DIS
LIN {X -85.1799,Y -96.0634,Z 141,A -135.2654,B 24.9648,C -1.3714,E1 24.893,E2 581.7433} C_DIS
LIN {X -88.4049,Y -93.1047,Z 141,A -137.2557,B 24.9647,C -1.3737,E1 24.8889,E2 583.7363} C_DIS
LIN {X -91.3709,Y -90.1958,Z 141,A -139.0667,B 24.9643,C -1.3797,E1 24.8854,E2 585.5406} C_DIS
LIN {X -94.2058,Y -87.2304,Z 141,A -140.9229,B 24.9642,C -1.3827,E1 24.8818,E2 587.3979} C_DIS
LIN {X -97.0105,Y -84.1004,Z 141,A -142.8646,B 24.9642,C -1.3839,E1 24.8782,E2 589.3454} C_DIS
LIN {X -99.7937,Y -80.7775,Z 141,A -144.7854,B 24.9639,C -1.3892,E1 24.8748,E2 591.2625} C_DIS
LIN {X -102.3497,Y -77.5134,Z 141,A -146.657,B 24.9637,C -1.3927,E1 24.8716,E2 593.1345} C_DIS
LIN {X -104.9903,Y -73.8972,Z 141,A -148.59,B 24.9632,C -1.4009,E1 24.8685,E2 595.0576} C_DIS
LIN {X -107.3566,Y -70.4156,Z 141,A -150.521,B 24.9632,C -1.4033,E1 24.8655,E2 596.9924} C_DIS
LIN {X -109.6518,Y -66.7862,Z 141,A -152.4949,B 24.963,C -1.4058,E1 24.8626,E2 598.9705} C_DIS
LIN {X -111.8301,Y -63.0698,Z 141,A -154.4031,B 24.9627,C -1.4117,E1 24.8599,E2 600.8745} C_DIS
LIN {X -113.7804,Y -59.4754,Z 141,A -156.1338,B 24.9622,C -1.4212,E1 24.8576,E2 602.5917} C_DIS
LIN {X -115.3046,Y -56.4646,Z 141,A -157.6807,B 24.962,C -1.4236,E1 24.8557,E2 604.1413} C_DIS
LIN {X -116.6449,Y -53.6406,Z 141,A -159.0775,B 24.9618,C -1.4276,E1 24.8541,E2 605.5363} C_DIS
LIN {X -117.9507,Y -50.7048,Z 141,A -160.497,B 24.9616,C -1.4324,E1 24.8525,E2 606.952} C_DIS
LIN {X -119.2143,Y -47.6589,Z 141,A -161.9663,B 24.9613,C -1.4369,E1 24.8509,E2 608.419} C_DIS
LIN {X -120.5086,Y -44.2898,Z 141,A -163.5857,B 24.9611,C -1.4413,E1 24.8493,E2 610.037} C_DIS
LIN {X -121.8819,Y -40.3504,Z 141,A -165.4751,B 24.9608,C -1.4457,E1 24.8476,E2 611.9266} C_DIS
LIN {X -122.9518,Y -36.9669,Z 141,A -167.0249,B 24.9605,C -1.4521,E1 24.8464,E2 613.47} C_DIS
LIN {X -123.7382,Y -34.2387,Z 141,A -168.2871,B 24.9603,C -1.4563,E1 24.8454,E2 614.7295} C_DIS
LIN {X -124.494,Y -31.3784,Z 141,A -169.6665,B 24.9602,C -1.4577,E1 24.8444,E2 616.1137} C_DIS
LIN {X -125.3182,Y -27.9133,Z 141,A -171.2491,B 24.9599,C -1.463,E1 24.8434,E2 617.6929} C_DIS
LIN {X -126.0454,Y -24.4131,Z 141,A -172.9108,B 24.9598,C -1.465,E1 24.8425,E2 619.3596} C_DIS
LIN {X -126.6499,Y -21.0514,Z 141,A -174.4241,B 24.9595,C -1.4704,E1 24.8418,E2 620.869} C_DIS
LIN {X -127.1573,Y -17.7356,Z 141,A -175.8601,B 24.9591,C -1.478,E1 24.8412,E2 622.2954} C_DIS
LIN {X -127.5059,Y -15.0212,Z 141,A -177.1761,B 24.9591,C -1.4777,E1 24.8408,E2 623.6202} C_DIS
LIN {X -127.9219,Y -10.9257,Z 141,A -179.0127,B 24.9588,C -1.4837,E1 24.8403,E2 625.4535} C_DIS
LIN {X -128.155,Y -7.7279,Z 141,A 179.566,B 24.9585,C -1.4888,E1 24.84,E2 626.8712} C_DIS
LIN {X -128.2983,Y -4.794,Z 141,A 178.3156,B 24.9581,C -1.4958,E1 24.8399,E2 628.1123} C_DIS
LIN {X -128.3763,Y -1.7531,Z 141,A 176.9528,B 24.9578,C -1.5,E1 24.8398,E2 629.4733} C_DIS
LIN {X -128.3702,Y 2.1225,Z 141,A 175.1244,B 24.9578,C -1.5012,E1 24.8398,E2 631.3099} C_DIS
LIN {X -128.262,Y 5.7236,Z 141,A 173.4272,B 24.9578,C -1.5024,E1 24.84,E2 633.0145} C_DIS
LIN {X -128.0509,Y 9.2923,Z 141,A 171.9324,B 24.9572,C -1.5123,E1 24.8403,E2 634.4947} C_DIS
LIN {X -127.7779,Y 12.4997,Z 141,A 170.4876,B 24.9569,C -1.5166,E1 24.8406,E2 635.9378} C_DIS
LIN {X -127.4432,Y 15.5471,Z 141,A 169.1515,B 24.9566,C -1.5226,E1 24.8411,E2 637.2677} C_DIS
LIN {X -127.0477,Y 18.503,Z 141,A 167.762,B 24.9565,C -1.5243,E1 24.8416,E2 638.6616} C_DIS
LIN {X -126.5797,Y 21.4719,Z 141,A 166.4011,B 24.9563,C -1.5277,E1 24.8422,E2 640.0222} C_DIS
LIN {X -126.0693,Y 24.2879,Z 141,A 165.0805,B 24.9561,C -1.5299,E1 24.8429,E2 641.3454} C_DIS
LIN {X -125.4426,Y 27.3413,Z 141,A 163.735,B 24.9558,C -1.5366,E1 24.8437,E2 642.683} C_DIS
LIN {X -124.7341,Y 30.411,Z 141,A 162.2837,B 24.9556,C -1.539,E1 24.8446,E2 644.137} C_DIS
LIN {X -123.9473,Y 33.4747,Z 141,A 160.8958,B 24.9553,C -1.5447,E1 24.8456,E2 645.5195} C_DIS
LIN {X -123.1513,Y 36.2919,Z 141,A 159.5487,B 24.9552,C -1.547,E1 24.8466,E2 646.8688} C_DIS
LIN {X -122.0599,Y 39.8158,Z 141,A 157.9072,B 24.9548,C -1.5525,E1 24.848,E2 648.5067} C_DIS
LIN {X -121.1149,Y 42.6006,Z 141,A 156.6063,B 24.9546,C -1.5572,E1 24.8492,E2 649.8038} C_DIS
LIN {X -120.1688,Y 45.197,Z 141,A 155.3205,B 24.9545,C -1.5587,E1 24.8504,E2 651.0932} C_DIS
LIN {X -118.8899,Y 48.4635,Z 141,A 153.7441,B 24.9542,C -1.5631,E1 24.8521,E2 652.6681} C_DIS
LIN {X -117.5976,Y 51.5216,Z 141,A 152.2835,B 24.9539,C -1.5686,E1 24.8537,E2 654.1235} C_DIS
LIN {X -116.394,Y 54.1831,Z 141,A 150.9514,B 24.9537,C -1.5713,E1 24.8552,E2 655.4564} C_DIS
LIN {X -114.9555,Y 57.1722,Z 141,A 149.4693,B 24.9535,C -1.5757,E1 24.857,E2 656.936} C_DIS
LIN {X -113.2348,Y 60.512,Z 141,A 147.6434,B 24.9535,C -1.5739,E1 24.8594,E2 658.7759} C_DIS
LIN {X -111.019,Y 64.4869,Z 141,A 145.6428,B 24.9531,C -1.5813,E1 24.8622,E2 660.7694} C_DIS
LIN {X -108.79,Y 68.181,Z 141,A 143.6594,B 24.953,C -1.5842,E1 24.8651,E2 662.756} C_DIS
LIN {X -106.4279,Y 71.8114,Z 141,A 141.7371,B 24.9526,C -1.5902,E1 24.868,E2 664.6736} C_DIS
LIN {X -103.8445,Y 75.499,Z 141,A 139.734,B 24.9523,C -1.5961,E1 24.8713,E2 666.6724} C_DIS
LIN {X -101.2232,Y 78.9796,Z 141,A 137.7756,B 24.952,C -1.6008,E1 24.8746,E2 668.6291} C_DIS
LIN {X -98.6224,Y 82.2042,Z 141,A 135.8733,B 24.9518,C -1.6033,E1 24.878,E2 670.5344} C_DIS
LIN {X -95.915,Y 85.3477,Z 141,A 134.011,B 24.9516,C -1.6076,E1 24.8814,E2 672.3948} C_DIS
LIN {X -93.1047,Y 88.4049,Z 141,A 132.2144,B 24.9511,C -1.6149,E1 24.8848,E2 674.1818} C_DIS
LIN {X -90.1958,Y 91.3709,Z 141,A 130.3581,B 24.9509,C -1.6194,E1 24.8885,E2 676.0353} C_DIS
LIN {X -87.1927,Y 94.2409,Z 141,A 128.4731,B 24.9507,C -1.6224,E1 24.8923,E2 677.9209} C_DIS
LIN {X -84.1004,Y 97.0105,Z 141,A 126.5592,B 24.9506,C -1.6238,E1 24.8963,E2 679.8389} C_DIS
LIN {X -80.9238,Y 99.6757,Z 141,A 124.6915,B 24.9504,C -1.6272,E1 24.9003,E2 681.7058} C_DIS
LIN {X -77.531,Y 102.3364,Z 141,A 122.78,B 24.9501,C -1.6319,E1 24.9046,E2 683.6129} C_DIS
LIN {X -73.9938,Y 104.9221,Z 141,A 120.8804,B 24.9497,C -1.6386,E1 24.9088,E2 685.5032} C_DIS
LIN {X -70.485,Y 107.3109,Z 141,A 118.9632,B 24.9495,C -1.6413,E1 24.9133,E2 687.4203} C_DIS
LIN {X -66.7862,Y 109.6518,Z 141,A 116.9453,B 24.9495,C -1.642,E1 24.9181,E2 689.443} C_DIS
LIN {X -63.0698,Y 111.8301,Z 141,A 115.0421,B 24.9492,C -1.6464,E1 24.9227,E2 691.3414} C_DIS
LIN {X -59.2493,Y 113.8991,Z 141,A 113.2212,B 24.9487,C -1.6553,E1 24.9271,E2 693.1462} C_DIS
LIN {X -56.504,Y 115.2852,Z 141,A 111.7839,B 24.9487,C -1.6545,E1 24.9307,E2 694.5892} C_DIS
LIN {X -53.4817,Y 116.7184,Z 141,A 110.3469,B 24.9484,C -1.6595,E1 24.9344,E2 696.018} C_DIS
LIN {X -50.6126,Y 117.9906,Z 141,A 108.9416,B 24.9483,C -1.6613,E1 24.9379,E2 697.4222} C_DIS
Enddeposition()
END
